(* Visualisation visuTimetable
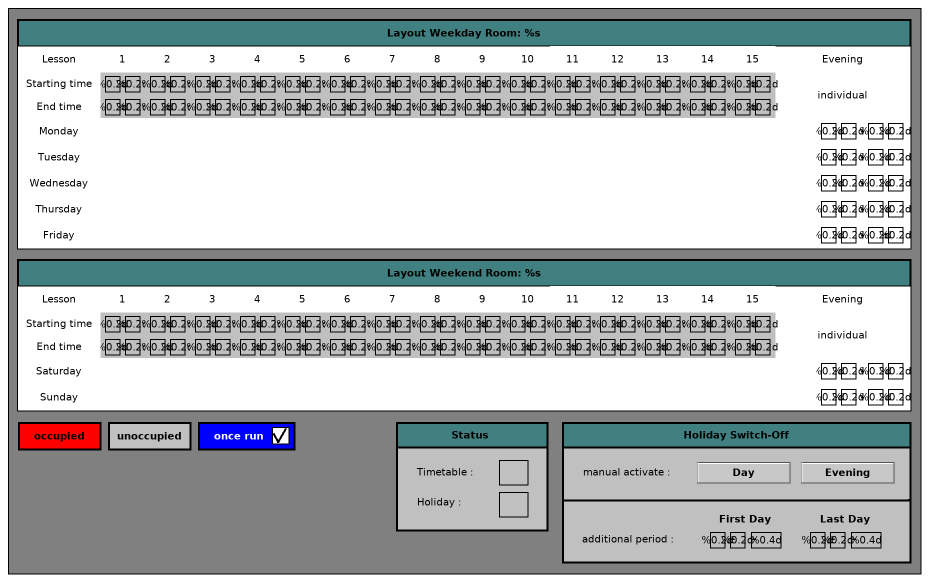
rectangle at (700,518)-(780,543): text "-     -"; tooltip First day Input format: DD-HH-YYYY
rectangle at (92,162)-(137,188): alarm colour if $typTimetable$.wDayLesson[3].1; toggles $typTimetable$.wDayLesson[3].1
rectangle at (137,162)-(182,188): alarm colour if $typTimetable$.wDayLesson[3].2; toggles $typTimetable$.wDayLesson[3].2
rectangle at (182,162)-(227,188): alarm colour if $typTimetable$.wDayLesson[3].3; toggles $typTimetable$.wDayLesson[3].3
rectangle at (227,162)-(272,188): alarm colour if $typTimetable$.wDayLesson[3].4; toggles $typTimetable$.wDayLesson[3].4
rectangle at (272,162)-(317,188): alarm colour if $typTimetable$.wDayLesson[3].5; toggles $typTimetable$.wDayLesson[3].5
rectangle at (317,162)-(362,188): alarm colour if $typTimetable$.wDayLesson[3].6; toggles $typTimetable$.wDayLesson[3].6
rectangle at (362,162)-(407,188): alarm colour if $typTimetable$.wDayLesson[3].7; toggles $typTimetable$.wDayLesson[3].7
rectangle at (407,162)-(452,188): alarm colour if $typTimetable$.wDayLesson[3].8; toggles $typTimetable$.wDayLesson[3].8
rectangle at (452,162)-(497,188): alarm colour if $typTimetable$.wDayLesson[3].9; toggles $typTimetable$.wDayLesson[3].9
rectangle at (497,162)-(542,188): alarm colour if $typTimetable$.wDayLesson[3].10; toggles $typTimetable$.wDayLesson[3].10
rectangle at (808,110)-(853,136): text ":"; tooltip Switch ON time of the scheduler single weekly
rectangle at (855,110)-(900,136): text ":"; tooltip Switch ON time of the scheduler single weekly
rectangle at (808,136)-(853,162): text ":"; tooltip Switch ON time of the scheduler single weekly
rectangle at (855,136)-(900,162): text ":"; tooltip Switch ON time of the scheduler single weekly
rectangle at (808,162)-(853,188): text ":"; tooltip Switch ON time of the scheduler single weekly
rectangle at (855,162)-(900,188): text ":"; tooltip Switch ON time of the scheduler single weekly
rectangle at (808,188)-(853,214): text ":"; tooltip Switch ON time of the scheduler single weekly
rectangle at (855,188)-(900,214): text ":"; tooltip Switch ON time of the scheduler single weekly
rectangle at (808,214)-(853,240): text ":"; tooltip Switch ON time of the scheduler single weekly
rectangle at (808,350)-(853,376): text ":"; tooltip Switch ON time of the scheduler single weekly
rectangle at (855,350)-(900,376): text ":"; tooltip Switch ON time of the scheduler single weekly
rectangle at (808,376)-(853,402): text ":"; tooltip Switch ON time of the scheduler single weekly
rectangle at (855,376)-(900,402): text ":"; tooltip Switch ON time of the scheduler single weekly
rectangle at (92,64)-(137,87): text ":"; tooltip Switch ON time
rectangle at (97,68)-(112,84): text "%0.2d"; shows $typLesson$.wWeekdayOn_hour[1]
rectangle at (117,68)-(132,84): text "%0.2d"; shows $typLesson$.wWeekdayOn_Minute[1]
rectangle at (137,64)-(182,87): text ":"; tooltip Switch ON time
rectangle at (142,68)-(157,84): text "%0.2d"; shows $typLesson$.wWeekdayOn_hour[2]
rectangle at (162,68)-(177,84): text "%0.2d"; shows $typLesson$.wWeekdayOn_Minute[2]
rectangle at (182,64)-(227,87): text ":"; tooltip Switch ON time
rectangle at (187,68)-(202,84): text "%0.2d"; shows $typLesson$.wWeekdayOn_hour[3]
rectangle at (207,68)-(222,84): text "%0.2d"; shows $typLesson$.wWeekdayOn_Minute[3]
rectangle at (227,64)-(272,87): text ":"; tooltip Switch ON time
rectangle at (232,68)-(247,84): text "%0.2d"; shows $typLesson$.wWeekdayOn_hour[4]
rectangle at (252,68)-(267,84): text "%0.2d"; shows $typLesson$.wWeekdayOn_Minute[4]
rectangle at (272,64)-(317,87): text ":"; tooltip Switch ON time
rectangle at (277,68)-(292,84): text "%0.2d"; shows $typLesson$.wWeekdayOn_hour[5]
rectangle at (297,68)-(312,84): text "%0.2d"; shows $typLesson$.wWeekdayOn_Minute[5]
rectangle at (317,64)-(362,87): text ":"; tooltip Switch ON time
rectangle at (322,68)-(337,84): text "%0.2d"; shows $typLesson$.wWeekdayOn_hour[6]
rectangle at (342,68)-(357,84): text "%0.2d"; shows $typLesson$.wWeekdayOn_Minute[6]
rectangle at (362,64)-(407,87): text ":"; tooltip Switch ON time
rectangle at (367,68)-(382,84): text "%0.2d"; shows $typLesson$.wWeekdayOn_hour[7]
rectangle at (387,68)-(402,84): text "%0.2d"; shows $typLesson$.wWeekdayOn_Minute[7]
rectangle at (407,64)-(452,87): text ":"; tooltip Switch ON time
rectangle at (412,68)-(427,84): text "%0.2d"; shows $typLesson$.wWeekdayOn_hour[8]
rectangle at (432,68)-(447,84): text "%0.2d"; shows $typLesson$.wWeekdayOn_Minute[8]
rectangle at (452,64)-(497,87): text ":"; tooltip Switch ON time
rectangle at (457,68)-(472,84): text "%0.2d"; shows $typLesson$.wWeekdayOn_hour[9]
rectangle at (477,68)-(492,84): text "%0.2d"; shows $typLesson$.wWeekdayOn_Minute[9]
rectangle at (497,64)-(542,87): text ":"; tooltip Switch ON time
rectangle at (502,68)-(517,84): text "%0.2d"; shows $typLesson$.wWeekdayOn_hour[10]
rectangle at (522,68)-(537,84): text "%0.2d"; shows $typLesson$.wWeekdayOn_Minute[10]
rectangle at (92,188)-(137,214): alarm colour if $typTimetable$.wDayLesson[4].1; toggles $typTimetable$.wDayLesson[4].1
rectangle at (137,188)-(182,214): alarm colour if $typTimetable$.wDayLesson[4].2; toggles $typTimetable$.wDayLesson[4].2
rectangle at (182,188)-(227,214): alarm colour if $typTimetable$.wDayLesson[4].3; toggles $typTimetable$.wDayLesson[4].3
rectangle at (227,188)-(272,214): alarm colour if $typTimetable$.wDayLesson[4].4; toggles $typTimetable$.wDayLesson[4].4
rectangle at (272,188)-(317,214): alarm colour if $typTimetable$.wDayLesson[4].5; toggles $typTimetable$.wDayLesson[4].5
rectangle at (317,188)-(362,214): alarm colour if $typTimetable$.wDayLesson[4].6; toggles $typTimetable$.wDayLesson[4].6
rectangle at (362,188)-(407,214): alarm colour if $typTimetable$.wDayLesson[4].7; toggles $typTimetable$.wDayLesson[4].7
rectangle at (407,188)-(452,214): alarm colour if $typTimetable$.wDayLesson[4].8; toggles $typTimetable$.wDayLesson[4].8
rectangle at (452,188)-(497,214): alarm colour if $typTimetable$.wDayLesson[4].9; toggles $typTimetable$.wDayLesson[4].9
rectangle at (497,188)-(542,214): alarm colour if $typTimetable$.wDayLesson[4].10; toggles $typTimetable$.wDayLesson[4].10
rectangle at (807,188)-(902,214): text "-"
rectangle at (807,214)-(902,240): text "-"
rectangle at (807,162)-(902,188): text "-"
rectangle at (807,136)-(902,162): text "-"
rectangle at (807,110)-(902,136): text "-"
rectangle at (813,115)-(828,131): text "%0.2d"; shows $typTimetable$.wEveningOn_hour[1]; editable 0..23
rectangle at (833,115)-(848,131): text "%0.2d"; shows $typTimetable$.wEveningOn_minute[1]; editable 0..59
rectangle at (860,115)-(875,131): text "%0.2d"; shows $typTimetable$.wEveningOff_hour[1]; editable 0..23
rectangle at (880,115)-(895,131): text "%0.2d"; shows $typTimetable$.wEveningOff_minute[1]; editable 0..59
rectangle at (813,141)-(828,157): text "%0.2d"; shows $typTimetable$.wEveningOn_hour[2]; editable 0..23
rectangle at (833,141)-(848,157): text "%0.2d"; shows $typTimetable$.wEveningOn_minute[2]; editable 0..59
rectangle at (860,141)-(875,157): text "%0.2d"; shows $typTimetable$.wEveningOff_hour[2]; editable 0..23
rectangle at (880,141)-(895,157): text "%0.2d"; shows $typTimetable$.wEveningOff_minute[2]; editable 0..59
rectangle at (813,193)-(828,209): text "%0.2d"; shows $typTimetable$.wEveningOn_hour[4]; editable 0..23
rectangle at (833,193)-(848,209): text "%0.2d"; shows $typTimetable$.wEveningOn_minute[4]; editable 0..59
rectangle at (860,193)-(875,209): text "%0.2d"; shows $typTimetable$.wEveningOff_hour[4]; editable 0..23
rectangle at (880,193)-(895,209): text "%0.2d"; shows $typTimetable$.wEveningOff_minute[4]; editable 0..59
rectangle at (813,219)-(828,235): text "%0.2d"; shows $typTimetable$.wEveningOn_hour[5]; editable 0..23
rectangle at (833,219)-(848,235): text "%0.2d"; shows $typTimetable$.wEveningOn_minute[5]; editable 0..59
rectangle at (813,167)-(828,183): text "%0.2d"; shows $typTimetable$.wEveningOn_hour[3]; editable 0..23
rectangle at (833,167)-(848,183): text "%0.2d"; shows $typTimetable$.wEveningOn_minute[3]; editable 0..59
rectangle at (860,167)-(875,183): text "%0.2d"; shows $typTimetable$.wEveningOff_hour[3]; editable 0..23
rectangle at (880,167)-(895,183): text "%0.2d"; shows $typTimetable$.wEveningOff_minute[3]; editable 0..59
rectangle at (807,350)-(902,376): text "-"
rectangle at (807,376)-(902,402): text "-"
rectangle at (813,355)-(828,371): text "%0.2d"; shows $typTimetable$.wEveningOn_hour[6]; editable 0..23
rectangle at (833,355)-(848,371): text "%0.2d"; shows $typTimetable$.wEveningOn_minute[6]; editable 0..59
rectangle at (860,355)-(875,371): text "%0.2d"; shows $typTimetable$.wEveningOff_hour[6]; editable 0..23
rectangle at (880,355)-(895,371): text "%0.2d"; shows $typTimetable$.wEveningOff_minute[6]; editable 0..59
rectangle at (813,381)-(828,397): text "%0.2d"; shows $typTimetable$.wEveningOn_hour[7]; editable 0..23
rectangle at (833,381)-(848,397): text "%0.2d"; shows $typTimetable$.wEveningOn_minute[7]; editable 0..59
rectangle at (860,381)-(875,397): text "%0.2d"; shows $typTimetable$.wEveningOff_hour[7]; editable 0..23
rectangle at (880,381)-(895,397): text "%0.2d"; shows $typTimetable$.wEveningOff_minute[7]; editable 0..59
rectangle at (92,110)-(137,136): alarm colour if $typTimetable$.wDayLesson[1].1; toggles $typTimetable$.wDayLesson[1].1
rectangle at (137,110)-(182,136): alarm colour if $typTimetable$.wDayLesson[1].2; toggles $typTimetable$.wDayLesson[1].2
rectangle at (182,110)-(227,136): alarm colour if $typTimetable$.wDayLesson[1].3; toggles $typTimetable$.wDayLesson[1].3
rectangle at (227,110)-(272,136): alarm colour if $typTimetable$.wDayLesson[1].4; toggles $typTimetable$.wDayLesson[1].4
rectangle at (272,110)-(317,136): alarm colour if $typTimetable$.wDayLesson[1].5; toggles $typTimetable$.wDayLesson[1].5
rectangle at (317,110)-(362,136): alarm colour if $typTimetable$.wDayLesson[1].6; toggles $typTimetable$.wDayLesson[1].6
rectangle at (362,110)-(407,136): alarm colour if $typTimetable$.wDayLesson[1].7; toggles $typTimetable$.wDayLesson[1].7
rectangle at (407,110)-(452,136): alarm colour if $typTimetable$.wDayLesson[1].8; toggles $typTimetable$.wDayLesson[1].8
rectangle at (452,110)-(497,136): alarm colour if $typTimetable$.wDayLesson[1].9; toggles $typTimetable$.wDayLesson[1].9
rectangle at (497,110)-(542,136): alarm colour if $typTimetable$.wDayLesson[1].10; toggles $typTimetable$.wDayLesson[1].10
rectangle at (92,136)-(137,162): alarm colour if $typTimetable$.wDayLesson[2].1; toggles $typTimetable$.wDayLesson[2].1
rectangle at (137,136)-(182,162): alarm colour if $typTimetable$.wDayLesson[2].2; toggles $typTimetable$.wDayLesson[2].2
rectangle at (182,136)-(227,162): alarm colour if $typTimetable$.wDayLesson[2].3; toggles $typTimetable$.wDayLesson[2].3
rectangle at (227,136)-(272,162): alarm colour if $typTimetable$.wDayLesson[2].4; toggles $typTimetable$.wDayLesson[2].4
rectangle at (272,136)-(317,162): alarm colour if $typTimetable$.wDayLesson[2].5; toggles $typTimetable$.wDayLesson[2].5
rectangle at (317,136)-(362,162): alarm colour if $typTimetable$.wDayLesson[2].6; toggles $typTimetable$.wDayLesson[2].6
rectangle at (362,136)-(407,162): alarm colour if $typTimetable$.wDayLesson[2].7; toggles $typTimetable$.wDayLesson[2].7
rectangle at (407,136)-(452,162): alarm colour if $typTimetable$.wDayLesson[2].8; toggles $typTimetable$.wDayLesson[2].8
rectangle at (452,136)-(497,162): alarm colour if $typTimetable$.wDayLesson[2].9; toggles $typTimetable$.wDayLesson[2].9
rectangle at (497,136)-(542,162): alarm colour if $typTimetable$.wDayLesson[2].10; toggles $typTimetable$.wDayLesson[2].10
rectangle at (92,214)-(137,240): alarm colour if $typTimetable$.wDayLesson[5].1; toggles $typTimetable$.wDayLesson[5].1
rectangle at (137,214)-(182,240): alarm colour if $typTimetable$.wDayLesson[5].2; toggles $typTimetable$.wDayLesson[5].2
rectangle at (182,214)-(227,240): alarm colour if $typTimetable$.wDayLesson[5].3; toggles $typTimetable$.wDayLesson[5].3
rectangle at (227,214)-(272,240): alarm colour if $typTimetable$.wDayLesson[5].4; toggles $typTimetable$.wDayLesson[5].4
rectangle at (272,214)-(317,240): alarm colour if $typTimetable$.wDayLesson[5].5; toggles $typTimetable$.wDayLesson[5].5
rectangle at (317,214)-(362,240): alarm colour if $typTimetable$.wDayLesson[5].6; toggles $typTimetable$.wDayLesson[5].6
rectangle at (362,214)-(407,240): alarm colour if $typTimetable$.wDayLesson[5].7; toggles $typTimetable$.wDayLesson[5].7
rectangle at (407,214)-(452,240): alarm colour if $typTimetable$.wDayLesson[5].8; toggles $typTimetable$.wDayLesson[5].8
rectangle at (452,214)-(497,240): alarm colour if $typTimetable$.wDayLesson[5].9; toggles $typTimetable$.wDayLesson[5].9
rectangle at (497,214)-(542,240): alarm colour if $typTimetable$.wDayLesson[5].10; toggles $typTimetable$.wDayLesson[5].10
rectangle at (92,350)-(137,376): alarm colour if $typTimetable$.wDayLesson[6].1; toggles $typTimetable$.wDayLesson[6].1
rectangle at (137,350)-(182,376): alarm colour if $typTimetable$.wDayLesson[6].2; toggles $typTimetable$.wDayLesson[6].2
rectangle at (182,350)-(227,376): alarm colour if $typTimetable$.wDayLesson[6].3; toggles $typTimetable$.wDayLesson[6].3
rectangle at (227,350)-(272,376): alarm colour if $typTimetable$.wDayLesson[6].4; toggles $typTimetable$.wDayLesson[6].4
rectangle at (272,350)-(317,376): alarm colour if $typTimetable$.wDayLesson[6].5; toggles $typTimetable$.wDayLesson[6].5
rectangle at (317,350)-(362,376): alarm colour if $typTimetable$.wDayLesson[6].6; toggles $typTimetable$.wDayLesson[6].6
rectangle at (362,350)-(407,376): alarm colour if $typTimetable$.wDayLesson[6].7; toggles $typTimetable$.wDayLesson[6].7
rectangle at (407,350)-(452,376): alarm colour if $typTimetable$.wDayLesson[6].8; toggles $typTimetable$.wDayLesson[6].8
rectangle at (452,350)-(497,376): alarm colour if $typTimetable$.wDayLesson[6].9; toggles $typTimetable$.wDayLesson[6].9
rectangle at (497,350)-(542,376): alarm colour if $typTimetable$.wDayLesson[6].10; toggles $typTimetable$.wDayLesson[6].10
rectangle at (92,376)-(137,402): alarm colour if $typTimetable$.wDayLesson[7].1; toggles $typTimetable$.wDayLesson[7].1
rectangle at (137,376)-(182,402): alarm colour if $typTimetable$.wDayLesson[7].2; toggles $typTimetable$.wDayLesson[7].2
rectangle at (182,376)-(227,402): alarm colour if $typTimetable$.wDayLesson[7].3; toggles $typTimetable$.wDayLesson[7].3
rectangle at (227,376)-(272,402): alarm colour if $typTimetable$.wDayLesson[7].4; toggles $typTimetable$.wDayLesson[7].4
rectangle at (272,376)-(317,402): alarm colour if $typTimetable$.wDayLesson[7].5; toggles $typTimetable$.wDayLesson[7].5
rectangle at (317,376)-(362,402): alarm colour if $typTimetable$.wDayLesson[7].6; toggles $typTimetable$.wDayLesson[7].6
rectangle at (362,376)-(407,402): alarm colour if $typTimetable$.wDayLesson[7].7; toggles $typTimetable$.wDayLesson[7].7
rectangle at (407,376)-(452,402): alarm colour if $typTimetable$.wDayLesson[7].8; toggles $typTimetable$.wDayLesson[7].8
rectangle at (452,376)-(497,402): alarm colour if $typTimetable$.wDayLesson[7].9; toggles $typTimetable$.wDayLesson[7].9
rectangle at (497,376)-(542,402): alarm colour if $typTimetable$.wDayLesson[7].10; toggles $typTimetable$.wDayLesson[7].10
rectangle at (92,87)-(137,110): text ":"; tooltip Switch OFF time
rectangle at (97,91)-(112,107): text "%0.2d"; shows $typLesson$.wWeekdayOff_hour[1]
rectangle at (117,91)-(132,107): text "%0.2d"; shows $typLesson$.wWeekdayOff_Minute[1]
rectangle at (137,87)-(182,110): text ":"; tooltip Switch OFF time
rectangle at (142,91)-(157,107): text "%0.2d"; shows $typLesson$.wWeekdayOff_hour[2]
rectangle at (162,91)-(177,107): text "%0.2d"; shows $typLesson$.wWeekdayOff_Minute[2]
rectangle at (182,87)-(227,110): text ":"; tooltip Switch OFF time
rectangle at (187,91)-(202,107): text "%0.2d"; shows $typLesson$.wWeekdayOff_hour[3]
rectangle at (207,91)-(222,107): text "%0.2d"; shows $typLesson$.wWeekdayOff_Minute[3]
rectangle at (227,87)-(272,110): text ":"; tooltip Switch OFF time
rectangle at (232,91)-(247,107): text "%0.2d"; shows $typLesson$.wWeekdayOff_hour[4]
rectangle at (252,91)-(267,107): text "%0.2d"; shows $typLesson$.wWeekdayOff_Minute[4]
rectangle at (272,87)-(317,110): text ":"; tooltip Switch OFF time
rectangle at (277,91)-(292,107): text "%0.2d"; shows $typLesson$.wWeekdayOff_hour[5]
rectangle at (297,91)-(312,107): text "%0.2d"; shows $typLesson$.wWeekdayOff_Minute[5]
rectangle at (317,87)-(362,110): text ":"; tooltip Switch OFF time
rectangle at (322,91)-(337,107): text "%0.2d"; shows $typLesson$.wWeekdayOff_hour[6]
rectangle at (342,91)-(357,107): text "%0.2d"; shows $typLesson$.wWeekdayOff_Minute[6]
rectangle at (362,87)-(407,110): text ":"; tooltip Switch OFF time
rectangle at (367,91)-(382,107): text "%0.2d"; shows $typLesson$.wWeekdayOff_hour[7]
rectangle at (387,91)-(402,107): text "%0.2d"; shows $typLesson$.wWeekdayOff_Minute[7]
rectangle at (407,87)-(452,110): text ":"; tooltip Switch OFF time
rectangle at (412,91)-(427,107): text "%0.2d"; shows $typLesson$.wWeekdayOff_hour[8]
rectangle at (432,91)-(447,107): text "%0.2d"; shows $typLesson$.wWeekdayOff_Minute[8]
rectangle at (452,87)-(497,110): text ":"; tooltip Switch OFF time
rectangle at (457,91)-(472,107): text "%0.2d"; shows $typLesson$.wWeekdayOff_hour[9]
rectangle at (477,91)-(492,107): text "%0.2d"; shows $typLesson$.wWeekdayOff_Minute[9]
rectangle at (497,87)-(542,110): text ":"; tooltip Switch OFF time
rectangle at (502,91)-(517,107): text "%0.2d"; shows $typLesson$.wWeekdayOff_hour[10]
rectangle at (522,91)-(537,107): text "%0.2d"; shows $typLesson$.wWeekdayOff_Minute[10]
rectangle at (767,64)-(902,110): text "individual"
rectangle at (92,38)-(137,64): text "1"
rectangle at (137,38)-(182,64): text "2"
rectangle at (182,38)-(227,64): text "3"
rectangle at (227,38)-(272,64): text "4"
rectangle at (272,38)-(317,64): text "5"
rectangle at (317,38)-(362,64): text "6"
rectangle at (362,38)-(407,64): text "7"
rectangle at (407,38)-(452,64): text "8"
rectangle at (452,38)-(497,64): text "9"
rectangle at (497,38)-(542,64): text "10"
rectangle at (767,38)-(902,64): text "Evening"
rectangle at (10,38)-(92,64): text "Lesson"
rectangle at (10,64)-(92,87): text "Starting time"
rectangle at (10,87)-(92,110): text "End time"
rectangle at (10,110)-(92,136): text "Monday"
rectangle at (10,136)-(92,162): text "Tuesday"
rectangle at (10,162)-(92,188): text "Wednesday"
rectangle at (10,188)-(92,214): text "Thursday"
rectangle at (10,214)-(92,240): text "Friday"
rectangle at (10,350)-(92,376): text "Saturday"
rectangle at (10,376)-(92,402): text "Sunday"
rectangle at (92,304)-(137,327): text ":"; tooltip Switch ON time
rectangle at (97,308)-(112,324): text "%0.2d"; shows $typLesson$.wWeekendOn_hour[1]
rectangle at (117,308)-(132,324): text "%0.2d"; shows $typLesson$.wWeekendOn_Minute[1]
rectangle at (137,304)-(182,327): text ":"; tooltip Switch ON time
rectangle at (142,308)-(157,324): text "%0.2d"; shows $typLesson$.wWeekendOn_hour[2]
rectangle at (162,308)-(177,324): text "%0.2d"; shows $typLesson$.wWeekendOn_Minute[2]
rectangle at (182,304)-(227,327): text ":"; tooltip Switch ON time
rectangle at (187,308)-(202,324): text "%0.2d"; shows $typLesson$.wWeekendOn_hour[3]
rectangle at (207,308)-(222,324): text "%0.2d"; shows $typLesson$.wWeekendOn_Minute[3]
rectangle at (227,304)-(272,327): text ":"; tooltip Switch ON time
rectangle at (232,308)-(247,324): text "%0.2d"; shows $typLesson$.wWeekendOn_hour[4]
rectangle at (252,308)-(267,324): text "%0.2d"; shows $typLesson$.wWeekendOn_Minute[4]
rectangle at (272,304)-(317,327): text ":"; tooltip Switch ON time
rectangle at (277,308)-(292,324): text "%0.2d"; shows $typLesson$.wWeekendOn_hour[5]
rectangle at (297,308)-(312,324): text "%0.2d"; shows $typLesson$.wWeekendOn_Minute[5]
rectangle at (317,304)-(362,327): text ":"; tooltip Switch ON time
rectangle at (322,308)-(337,324): text "%0.2d"; shows $typLesson$.wWeekendOn_hour[6]
rectangle at (342,308)-(357,324): text "%0.2d"; shows $typLesson$.wWeekendOn_Minute[6]
rectangle at (362,304)-(407,327): text ":"; tooltip Switch ON time
rectangle at (367,308)-(382,324): text "%0.2d"; shows $typLesson$.wWeekendOn_hour[7]
rectangle at (387,308)-(402,324): text "%0.2d"; shows $typLesson$.wWeekendOn_Minute[7]
rectangle at (407,304)-(452,327): text ":"; tooltip Switch ON time
rectangle at (412,308)-(427,324): text "%0.2d"; shows $typLesson$.wWeekendOn_hour[8]
rectangle at (432,308)-(447,324): text "%0.2d"; shows $typLesson$.wWeekendOn_Minute[8]
rectangle at (452,304)-(497,327): text ":"; tooltip Switch ON time
rectangle at (457,308)-(472,324): text "%0.2d"; shows $typLesson$.wWeekendOn_hour[9]
rectangle at (477,308)-(492,324): text "%0.2d"; shows $typLesson$.wWeekendOn_Minute[9]
rectangle at (497,304)-(542,327): text ":"; tooltip Switch ON time
rectangle at (502,308)-(517,324): text "%0.2d"; shows $typLesson$.wWeekendOn_hour[10]
rectangle at (522,308)-(537,324): text "%0.2d"; shows $typLesson$.wWeekendOn_Minute[10]
rectangle at (92,327)-(137,350): text ":"; tooltip Switch OFF time
rectangle at (97,331)-(112,347): text "%0.2d"; shows $typLesson$.wWeekendOff_hour[1]
rectangle at (117,331)-(132,347): text "%0.2d"; shows $typLesson$.wWeekendOff_Minute[1]
rectangle at (137,327)-(182,350): text ":"; tooltip Switch OFF time
rectangle at (142,331)-(157,347): text "%0.2d"; shows $typLesson$.wWeekendOff_hour[2]
rectangle at (162,331)-(177,347): text "%0.2d"; shows $typLesson$.wWeekendOff_Minute[2]
rectangle at (182,327)-(227,350): text ":"; tooltip Switch OFF time
rectangle at (187,331)-(202,347): text "%0.2d"; shows $typLesson$.wWeekendOff_hour[3]
rectangle at (207,331)-(222,347): text "%0.2d"; shows $typLesson$.wWeekendOff_Minute[3]
rectangle at (227,327)-(272,350): text ":"; tooltip Switch OFF time
rectangle at (232,331)-(247,347): text "%0.2d"; shows $typLesson$.wWeekendOff_hour[4]
rectangle at (252,331)-(267,347): text "%0.2d"; shows $typLesson$.wWeekendOff_Minute[4]
rectangle at (272,327)-(317,350): text ":"; tooltip Switch OFF time
rectangle at (277,331)-(292,347): text "%0.2d"; shows $typLesson$.wWeekendOff_hour[5]
rectangle at (297,331)-(312,347): text "%0.2d"; shows $typLesson$.wWeekendOff_Minute[5]
rectangle at (317,327)-(362,350): text ":"; tooltip Switch OFF time
rectangle at (322,331)-(337,347): text "%0.2d"; shows $typLesson$.wWeekendOff_hour[6]
rectangle at (342,331)-(357,347): text "%0.2d"; shows $typLesson$.wWeekendOff_Minute[6]
rectangle at (362,327)-(407,350): text ":"; tooltip Switch OFF time
rectangle at (367,331)-(382,347): text "%0.2d"; shows $typLesson$.wWeekendOff_hour[7]
rectangle at (387,331)-(402,347): text "%0.2d"; shows $typLesson$.wWeekendOff_Minute[7]
rectangle at (407,327)-(452,350): text ":"; tooltip Switch OFF time
rectangle at (412,331)-(427,347): text "%0.2d"; shows $typLesson$.wWeekendOff_hour[8]
rectangle at (432,331)-(447,347): text "%0.2d"; shows $typLesson$.wWeekendOff_Minute[8]
rectangle at (452,327)-(497,350): text ":"; tooltip Switch OFF time
rectangle at (457,331)-(472,347): text "%0.2d"; shows $typLesson$.wWeekendOff_hour[9]
rectangle at (477,331)-(492,347): text "%0.2d"; shows $typLesson$.wWeekendOff_Minute[9]
rectangle at (497,327)-(542,350): text ":"; tooltip Switch OFF time
rectangle at (502,331)-(517,347): text "%0.2d"; shows $typLesson$.wWeekendOff_hour[10]
rectangle at (522,331)-(537,347): text "%0.2d"; shows $typLesson$.wWeekendOff_Minute[10]
rectangle at (767,304)-(902,350): text "individual"
rectangle at (92,278)-(137,304): text "1"
rectangle at (137,278)-(182,304): text "2"
rectangle at (182,278)-(227,304): text "3"
rectangle at (227,278)-(272,304): text "4"
rectangle at (272,278)-(317,304): text "5"
rectangle at (317,278)-(362,304): text "6"
rectangle at (362,278)-(407,304): text "7"
rectangle at (407,278)-(452,304): text "8"
rectangle at (452,278)-(497,304): text "9"
rectangle at (497,278)-(542,304): text "10"
rectangle at (767,278)-(902,304): text "Evening"
rectangle at (10,278)-(92,304): text "Lesson"
rectangle at (10,304)-(92,327): text "Starting time"
rectangle at (10,327)-(92,350): text "End time"
rectangle at (10,252)-(902,278): text "Layout Weekend Room: %s"; shows $typTimetable$.stRoomNr; editable
rectangle at (10,12)-(902,38): text "Layout Weekday Room: %s"; shows $typTimetable$.stRoomNr; editable
button at (689,454)-(782,475): text "Day"; toggles $typTimetable$.bConfig.0
button at (793,454)-(886,475): text "Evening"; toggles $typTimetable$.bConfig.1
rectangle at (554,414)-(903,440): text "Holiday Switch-Off"
rectangle at (10,414)-(93,442): text "occupied"
rectangle at (100,414)-(183,442): text "unoccupied"
rectangle at (542,162)-(587,188): alarm colour if $typTimetable$.wDayLesson[3].11; toggles $typTimetable$.wDayLesson[3].11
rectangle at (542,64)-(587,87): text ":"; tooltip Switch ON time
rectangle at (547,68)-(562,84): text "%0.2d"; shows $typLesson$.wWeekdayOn_hour[11]
rectangle at (567,68)-(582,84): text "%0.2d"; shows $typLesson$.wWeekdayOn_Minute[11]
rectangle at (542,188)-(587,214): alarm colour if $typTimetable$.wDayLesson[4].11; toggles $typTimetable$.wDayLesson[4].11
rectangle at (542,110)-(587,136): alarm colour if $typTimetable$.wDayLesson[1].11; toggles $typTimetable$.wDayLesson[1].11
rectangle at (542,136)-(587,162): alarm colour if $typTimetable$.wDayLesson[2].11; toggles $typTimetable$.wDayLesson[2].11
rectangle at (542,214)-(587,240): alarm colour if $typTimetable$.wDayLesson[5].11; toggles $typTimetable$.wDayLesson[5].11
rectangle at (542,87)-(587,110): text ":"; tooltip Switch OFF time
rectangle at (547,91)-(562,107): text "%0.2d"; shows $typLesson$.wWeekdayOff_hour[11]
rectangle at (567,91)-(582,107): text "%0.2d"; shows $typLesson$.wWeekdayOff_Minute[11]
rectangle at (542,38)-(587,64): text "11"
rectangle at (587,162)-(632,188): alarm colour if $typTimetable$.wDayLesson[3].12; toggles $typTimetable$.wDayLesson[3].12
rectangle at (587,64)-(632,87): text ":"; tooltip Switch ON time
rectangle at (592,68)-(607,84): text "%0.2d"; shows $typLesson$.wWeekdayOn_hour[12]
rectangle at (612,68)-(627,84): text "%0.2d"; shows $typLesson$.wWeekdayOn_Minute[12]
rectangle at (587,188)-(632,214): alarm colour if $typTimetable$.wDayLesson[4].12; toggles $typTimetable$.wDayLesson[4].12
rectangle at (587,110)-(632,136): alarm colour if $typTimetable$.wDayLesson[1].12; toggles $typTimetable$.wDayLesson[1].12
rectangle at (587,136)-(632,162): alarm colour if $typTimetable$.wDayLesson[2].12; toggles $typTimetable$.wDayLesson[2].12
rectangle at (587,214)-(632,240): alarm colour if $typTimetable$.wDayLesson[5].12; toggles $typTimetable$.wDayLesson[5].12
rectangle at (587,87)-(632,110): text ":"; tooltip Switch OFF time
rectangle at (592,91)-(607,107): text "%0.2d"; shows $typLesson$.wWeekdayOff_hour[12]
rectangle at (612,91)-(627,107): text "%0.2d"; shows $typLesson$.wWeekdayOff_Minute[12]
rectangle at (587,38)-(632,64): text "12"
rectangle at (632,162)-(677,188): alarm colour if $typTimetable$.wDayLesson[3].13; toggles $typTimetable$.wDayLesson[3].13
rectangle at (632,64)-(677,87): text ":"; tooltip Switch ON time
rectangle at (637,68)-(652,84): text "%0.2d"; shows $typLesson$.wWeekdayOn_hour[13]
rectangle at (657,68)-(672,84): text "%0.2d"; shows $typLesson$.wWeekdayOn_Minute[13]
rectangle at (632,188)-(677,214): alarm colour if $typTimetable$.wDayLesson[4].13; toggles $typTimetable$.wDayLesson[4].13
rectangle at (632,110)-(677,136): alarm colour if $typTimetable$.wDayLesson[1].13; toggles $typTimetable$.wDayLesson[1].13
rectangle at (632,136)-(677,162): alarm colour if $typTimetable$.wDayLesson[2].13; toggles $typTimetable$.wDayLesson[2].13
rectangle at (632,214)-(677,240): alarm colour if $typTimetable$.wDayLesson[5].13; toggles $typTimetable$.wDayLesson[5].13
rectangle at (632,87)-(677,110): text ":"; tooltip Switch OFF time
rectangle at (637,91)-(652,107): text "%0.2d"; shows $typLesson$.wWeekdayOff_hour[13]
rectangle at (657,91)-(672,107): text "%0.2d"; shows $typLesson$.wWeekdayOff_Minute[13]
rectangle at (632,38)-(677,64): text "13"
rectangle at (677,162)-(722,188): alarm colour if $typTimetable$.wDayLesson[3].14; toggles $typTimetable$.wDayLesson[3].14
rectangle at (677,64)-(722,87): text ":"; tooltip Switch ON time
rectangle at (682,68)-(697,84): text "%0.2d"; shows $typLesson$.wWeekdayOn_hour[14]
rectangle at (702,68)-(717,84): text "%0.2d"; shows $typLesson$.wWeekdayOn_Minute[14]
rectangle at (677,188)-(722,214): alarm colour if $typTimetable$.wDayLesson[4].14; toggles $typTimetable$.wDayLesson[4].14
rectangle at (677,110)-(722,136): alarm colour if $typTimetable$.wDayLesson[1].14; toggles $typTimetable$.wDayLesson[1].14
rectangle at (677,136)-(722,162): alarm colour if $typTimetable$.wDayLesson[2].14; toggles $typTimetable$.wDayLesson[2].14
rectangle at (677,214)-(722,240): alarm colour if $typTimetable$.wDayLesson[5].14; toggles $typTimetable$.wDayLesson[5].14
rectangle at (677,87)-(722,110): text ":"; tooltip Switch OFF time
rectangle at (682,91)-(697,107): text "%0.2d"; shows $typLesson$.wWeekdayOff_hour[14]
rectangle at (702,91)-(717,107): text "%0.2d"; shows $typLesson$.wWeekdayOff_Minute[14]
rectangle at (677,38)-(722,64): text "14"
rectangle at (722,162)-(767,188): alarm colour if $typTimetable$.wDayLesson[3].15; toggles $typTimetable$.wDayLesson[3].15
rectangle at (722,64)-(767,87): text ":"; tooltip Switch ON time
rectangle at (727,68)-(742,84): text "%0.2d"; shows $typLesson$.wWeekdayOn_hour[15]
rectangle at (747,68)-(762,84): text "%0.2d"; shows $typLesson$.wWeekdayOn_Minute[15]
rectangle at (722,188)-(767,214): alarm colour if $typTimetable$.wDayLesson[4].15; toggles $typTimetable$.wDayLesson[4].15
rectangle at (722,110)-(767,136): alarm colour if $typTimetable$.wDayLesson[1].15; toggles $typTimetable$.wDayLesson[1].15
rectangle at (722,136)-(767,162): alarm colour if $typTimetable$.wDayLesson[2].15; toggles $typTimetable$.wDayLesson[2].15
rectangle at (722,214)-(767,240): alarm colour if $typTimetable$.wDayLesson[5].15; toggles $typTimetable$.wDayLesson[5].15
rectangle at (722,87)-(767,110): text ":"; tooltip Switch OFF time
rectangle at (727,91)-(742,107): text "%0.2d"; shows $typLesson$.wWeekdayOff_hour[15]
rectangle at (747,91)-(762,107): text "%0.2d"; shows $typLesson$.wWeekdayOff_Minute[15]
rectangle at (722,38)-(767,64): text "15"
rectangle at (542,350)-(587,376): alarm colour if $typTimetable$.wDayLesson[6].11; toggles $typTimetable$.wDayLesson[6].11
rectangle at (542,376)-(587,402): alarm colour if $typTimetable$.wDayLesson[7].11; toggles $typTimetable$.wDayLesson[7].11
rectangle at (542,304)-(587,327): text ":"; tooltip Switch ON time
rectangle at (547,308)-(562,324): text "%0.2d"; shows $typLesson$.wWeekendOn_hour[11]
rectangle at (567,308)-(582,324): text "%0.2d"; shows $typLesson$.wWeekendOn_Minute[11]
rectangle at (542,327)-(587,350): text ":"; tooltip Switch OFF time
rectangle at (547,331)-(562,347): text "%0.2d"; shows $typLesson$.wWeekendOff_hour[11]
rectangle at (567,331)-(582,347): text "%0.2d"; shows $typLesson$.wWeekendOff_Minute[11]
rectangle at (542,278)-(587,304): text "11"
rectangle at (587,350)-(632,376): alarm colour if $typTimetable$.wDayLesson[6].12; toggles $typTimetable$.wDayLesson[6].12
rectangle at (587,376)-(632,402): alarm colour if $typTimetable$.wDayLesson[7].12; toggles $typTimetable$.wDayLesson[7].12
rectangle at (587,304)-(632,327): text ":"; tooltip Switch ON time
rectangle at (592,308)-(607,324): text "%0.2d"; shows $typLesson$.wWeekendOn_hour[12]
rectangle at (612,308)-(627,324): text "%0.2d"; shows $typLesson$.wWeekendOn_Minute[12]
rectangle at (587,327)-(632,350): text ":"; tooltip Switch OFF time
rectangle at (592,331)-(607,347): text "%0.2d"; shows $typLesson$.wWeekendOff_hour[12]
rectangle at (612,331)-(627,347): text "%0.2d"; shows $typLesson$.wWeekendOff_Minute[12]
rectangle at (587,278)-(632,304): text "12"
rectangle at (632,350)-(677,376): alarm colour if $typTimetable$.wDayLesson[6].13; toggles $typTimetable$.wDayLesson[6].13
rectangle at (632,376)-(677,402): alarm colour if $typTimetable$.wDayLesson[7].13; toggles $typTimetable$.wDayLesson[7].13
rectangle at (632,304)-(677,327): text ":"; tooltip Switch ON time
rectangle at (637,308)-(652,324): text "%0.2d"; shows $typLesson$.wWeekendOn_hour[13]
rectangle at (657,308)-(672,324): text "%0.2d"; shows $typLesson$.wWeekendOn_Minute[13]
rectangle at (632,327)-(677,350): text ":"; tooltip Switch OFF time
rectangle at (637,331)-(652,347): text "%0.2d"; shows $typLesson$.wWeekendOff_hour[13]
rectangle at (657,331)-(672,347): text "%0.2d"; shows $typLesson$.wWeekendOff_Minute[13]
rectangle at (632,278)-(677,304): text "13"
rectangle at (677,350)-(722,376): alarm colour if $typTimetable$.wDayLesson[6].14; toggles $typTimetable$.wDayLesson[6].14
rectangle at (677,376)-(722,402): alarm colour if $typTimetable$.wDayLesson[7].14; toggles $typTimetable$.wDayLesson[7].14
rectangle at (677,304)-(722,327): text ":"; tooltip Switch ON time
rectangle at (682,308)-(697,324): text "%0.2d"; shows $typLesson$.wWeekendOn_hour[14]
rectangle at (702,308)-(717,324): text "%0.2d"; shows $typLesson$.wWeekendOn_Minute[14]
rectangle at (677,327)-(722,350): text ":"; tooltip Switch OFF time
rectangle at (682,331)-(697,347): text "%0.2d"; shows $typLesson$.wWeekendOff_hour[14]
rectangle at (702,331)-(717,347): text "%0.2d"; shows $typLesson$.wWeekendOff_Minute[14]
rectangle at (677,278)-(722,304): text "14"
rectangle at (722,350)-(767,376): alarm colour if $typTimetable$.wDayLesson[6].15; toggles $typTimetable$.wDayLesson[6].15
rectangle at (722,376)-(767,402): alarm colour if $typTimetable$.wDayLesson[7].15; toggles $typTimetable$.wDayLesson[7].15
rectangle at (722,304)-(767,327): text ":"; tooltip Switch ON time
rectangle at (727,308)-(742,324): text "%0.2d"; shows $typLesson$.wWeekendOn_hour[15]
rectangle at (747,308)-(762,324): text "%0.2d"; shows $typLesson$.wWeekendOn_Minute[15]
rectangle at (722,327)-(767,350): text ":"; tooltip Switch OFF time
rectangle at (727,331)-(742,347): text "%0.2d"; shows $typLesson$.wWeekendOff_hour[15]
rectangle at (747,331)-(762,347): text "%0.2d"; shows $typLesson$.wWeekendOff_Minute[15]
rectangle at (722,278)-(767,304): text "15"
rectangle at (767,110)-(807,136): alarm colour if $typTimetable$.wDayLesson[1].0; toggles $typTimetable$.wDayLesson[1].0
rectangle at (767,136)-(807,162): alarm colour if $typTimetable$.wDayLesson[2].0; toggles $typTimetable$.wDayLesson[2].0
rectangle at (767,162)-(807,188): alarm colour if $typTimetable$.wDayLesson[3].0; toggles $typTimetable$.wDayLesson[3].0
rectangle at (767,188)-(807,214): alarm colour if $typTimetable$.wDayLesson[4].0; toggles $typTimetable$.wDayLesson[4].0
rectangle at (767,214)-(807,240): alarm colour if $typTimetable$.wDayLesson[5].0; toggles $typTimetable$.wDayLesson[5].0
rectangle at (767,350)-(807,376): alarm colour if $typTimetable$.wDayLesson[6].0; toggles $typTimetable$.wDayLesson[6].0
rectangle at (767,376)-(807,402): alarm colour if $typTimetable$.wDayLesson[7].0; toggles $typTimetable$.wDayLesson[7].0
rectangle at (800,518)-(880,543): text "-     -"; tooltip Last day Input format: DD-HH-YYYY
rectangle at (802,524)-(817,540): text "%0.2d"; shows $typTimetable$.wSpecialLastDay[1]; editable 0..31
rectangle at (822,524)-(837,540): text "%0.2d"; shows $typTimetable$.wSpecialLastDay[2]; editable 0..12
rectangle at (843,524)-(873,540): text "%0.4d"; shows $typTimetable$.wSpecialLastDay[3]; editable 0..2099
rectangle at (702,524)-(717,540): text "%0.2d"; shows $typTimetable$.wSpecialFirstDay[1]; editable 0..31
rectangle at (722,524)-(737,540): text "%0.2d"; shows $typTimetable$.wSpecialFirstDay[2]; editable 0..12
rectangle at (743,524)-(773,540): text "%0.4d"; shows $typTimetable$.wSpecialFirstDay[3]; editable 0..2099
rectangle at (388,414)-(540,440): text "Status"
rectangle at (395,451)-(480,477): text "Timetable :"
rectangle at (395,481)-(473,507): text "Holiday :"
rectangle at (561,451)-(689,477): text "manual activate :"
rectangle at (560,518)-(688,544): text "additional period :"
rectangle at (697,499)-(777,523): text "First Day"
rectangle at (797,499)-(877,523): text "Last Day"
rectangle at (491,452)-(520,477): alarm colour if $typTimetable$.bStatus.1
rectangle at (491,484)-(520,509): alarm colour if $typTimetable$.bStatus.2
rectangle at (92,110)-(137,136): invisible if NOT $typTimetable$.bConfig.2 AND NOT ($typTimetable$.wDayLessonOnce[1].1 AND NOT $typTimetable$.bConfig.2); alarm colour if $typTimetable$.wDayLessonOnce[1].1; toggles $typTimetable$.wDayLessonOnce[1].1
rectangle at (137,110)-(182,136): invisible if NOT $typTimetable$.bConfig.2 AND NOT ($typTimetable$.wDayLessonOnce[1].2 AND NOT $typTimetable$.bConfig.2); alarm colour if $typTimetable$.wDayLessonOnce[1].2; toggles $typTimetable$.wDayLessonOnce[1].2
rectangle at (182,110)-(227,136): invisible if NOT $typTimetable$.bConfig.2 AND NOT ($typTimetable$.wDayLessonOnce[1].3 AND NOT $typTimetable$.bConfig.2); alarm colour if $typTimetable$.wDayLessonOnce[1].3; toggles $typTimetable$.wDayLessonOnce[1].3
rectangle at (227,110)-(272,136): invisible if NOT $typTimetable$.bConfig.2 AND NOT ($typTimetable$.wDayLessonOnce[1].4 AND NOT $typTimetable$.bConfig.2); alarm colour if $typTimetable$.wDayLessonOnce[1].4; toggles $typTimetable$.wDayLessonOnce[1].4
rectangle at (272,110)-(317,136): invisible if NOT $typTimetable$.bConfig.2 AND NOT ($typTimetable$.wDayLessonOnce[1].5 AND NOT $typTimetable$.bConfig.2); alarm colour if $typTimetable$.wDayLessonOnce[1].5; toggles $typTimetable$.wDayLessonOnce[1].5
rectangle at (317,110)-(362,136): invisible if NOT $typTimetable$.bConfig.2 AND NOT ($typTimetable$.wDayLessonOnce[1].6 AND NOT $typTimetable$.bConfig.2); alarm colour if $typTimetable$.wDayLessonOnce[1].6; toggles $typTimetable$.wDayLessonOnce[1].6
rectangle at (362,110)-(407,136): invisible if NOT $typTimetable$.bConfig.2 AND NOT ($typTimetable$.wDayLessonOnce[1].7 AND NOT $typTimetable$.bConfig.2); alarm colour if $typTimetable$.wDayLessonOnce[1].7; toggles $typTimetable$.wDayLessonOnce[1].7
rectangle at (407,110)-(452,136): invisible if NOT $typTimetable$.bConfig.2 AND NOT ($typTimetable$.wDayLessonOnce[1].8 AND NOT $typTimetable$.bConfig.2); alarm colour if $typTimetable$.wDayLessonOnce[1].8; toggles $typTimetable$.wDayLessonOnce[1].8
rectangle at (452,110)-(497,136): invisible if NOT $typTimetable$.bConfig.2 AND NOT ($typTimetable$.wDayLessonOnce[1].9 AND NOT $typTimetable$.bConfig.2); alarm colour if $typTimetable$.wDayLessonOnce[1].9; toggles $typTimetable$.wDayLessonOnce[1].9
rectangle at (497,110)-(542,136): invisible if NOT $typTimetable$.bConfig.2 AND NOT ($typTimetable$.wDayLessonOnce[1].10 AND NOT $typTimetable$.bConfig.2); alarm colour if $typTimetable$.wDayLessonOnce[1].10; toggles $typTimetable$.wDayLessonOnce[1].10
rectangle at (542,110)-(587,136): invisible if NOT $typTimetable$.bConfig.2 AND NOT ($typTimetable$.wDayLessonOnce[1].11 AND NOT $typTimetable$.bConfig.2); alarm colour if $typTimetable$.wDayLessonOnce[1].11; toggles $typTimetable$.wDayLessonOnce[1].11
rectangle at (587,110)-(632,136): invisible if NOT $typTimetable$.bConfig.2 AND NOT ($typTimetable$.wDayLessonOnce[1].12 AND NOT $typTimetable$.bConfig.2); alarm colour if $typTimetable$.wDayLessonOnce[1].12; toggles $typTimetable$.wDayLessonOnce[1].12
rectangle at (632,110)-(677,136): invisible if NOT $typTimetable$.bConfig.2 AND NOT ($typTimetable$.wDayLessonOnce[1].13 AND NOT $typTimetable$.bConfig.2); alarm colour if $typTimetable$.wDayLessonOnce[1].13; toggles $typTimetable$.wDayLessonOnce[1].13
rectangle at (677,110)-(722,136): invisible if NOT $typTimetable$.bConfig.2 AND NOT ($typTimetable$.wDayLessonOnce[1].14 AND NOT $typTimetable$.bConfig.2); alarm colour if $typTimetable$.wDayLessonOnce[1].14; toggles $typTimetable$.wDayLessonOnce[1].14
rectangle at (722,110)-(767,136): invisible if NOT $typTimetable$.bConfig.2 AND NOT ($typTimetable$.wDayLessonOnce[1].15 AND NOT $typTimetable$.bConfig.2); alarm colour if $typTimetable$.wDayLessonOnce[1].15; toggles $typTimetable$.wDayLessonOnce[1].15
rectangle at (766,110)-(808,136): invisible if NOT $typTimetable$.bConfig.2 AND NOT ($typTimetable$.wDayLessonOnce[1].0 AND NOT $typTimetable$.bConfig.2); alarm colour if $typTimetable$.wDayLessonOnce[1].0; toggles $typTimetable$.wDayLessonOnce[1].0
rectangle at (92,136)-(137,162): invisible if NOT $typTimetable$.bConfig.2 AND NOT ($typTimetable$.wDayLessonOnce[2].1 AND NOT $typTimetable$.bConfig.2); alarm colour if $typTimetable$.wDayLessonOnce[2].1; toggles $typTimetable$.wDayLessonOnce[2].1
rectangle at (137,136)-(182,162): invisible if NOT $typTimetable$.bConfig.2 AND NOT ($typTimetable$.wDayLessonOnce[2].2 AND NOT $typTimetable$.bConfig.2); alarm colour if $typTimetable$.wDayLessonOnce[2].2; toggles $typTimetable$.wDayLessonOnce[2].2
rectangle at (182,136)-(227,162): invisible if NOT $typTimetable$.bConfig.2 AND NOT ($typTimetable$.wDayLessonOnce[2].3 AND NOT $typTimetable$.bConfig.2); alarm colour if $typTimetable$.wDayLessonOnce[2].3; toggles $typTimetable$.wDayLessonOnce[2].3
rectangle at (227,136)-(272,162): invisible if NOT $typTimetable$.bConfig.2 AND NOT ($typTimetable$.wDayLessonOnce[2].4 AND NOT $typTimetable$.bConfig.2); alarm colour if $typTimetable$.wDayLessonOnce[2].4; toggles $typTimetable$.wDayLessonOnce[2].4
rectangle at (272,136)-(317,162): invisible if NOT $typTimetable$.bConfig.2 AND NOT ($typTimetable$.wDayLessonOnce[2].5 AND NOT $typTimetable$.bConfig.2); alarm colour if $typTimetable$.wDayLessonOnce[2].5; toggles $typTimetable$.wDayLessonOnce[2].5
rectangle at (317,136)-(362,162): invisible if NOT $typTimetable$.bConfig.2 AND NOT ($typTimetable$.wDayLessonOnce[2].6 AND NOT $typTimetable$.bConfig.2); alarm colour if $typTimetable$.wDayLessonOnce[2].6; toggles $typTimetable$.wDayLessonOnce[2].6
rectangle at (362,136)-(407,162): invisible if NOT $typTimetable$.bConfig.2 AND NOT ($typTimetable$.wDayLessonOnce[2].7 AND NOT $typTimetable$.bConfig.2); alarm colour if $typTimetable$.wDayLessonOnce[2].7; toggles $typTimetable$.wDayLessonOnce[2].7
rectangle at (407,136)-(452,162): invisible if NOT $typTimetable$.bConfig.2 AND NOT ($typTimetable$.wDayLessonOnce[2].8 AND NOT $typTimetable$.bConfig.2); alarm colour if $typTimetable$.wDayLessonOnce[2].8; toggles $typTimetable$.wDayLessonOnce[2].8
rectangle at (452,136)-(497,162): invisible if NOT $typTimetable$.bConfig.2 AND NOT ($typTimetable$.wDayLessonOnce[2].9 AND NOT $typTimetable$.bConfig.2); alarm colour if $typTimetable$.wDayLessonOnce[2].9; toggles $typTimetable$.wDayLessonOnce[2].9
rectangle at (497,136)-(542,162): invisible if NOT $typTimetable$.bConfig.2 AND NOT ($typTimetable$.wDayLessonOnce[2].10 AND NOT $typTimetable$.bConfig.2); alarm colour if $typTimetable$.wDayLessonOnce[2].10; toggles $typTimetable$.wDayLessonOnce[2].10
rectangle at (542,136)-(587,162): invisible if NOT $typTimetable$.bConfig.2 AND NOT ($typTimetable$.wDayLessonOnce[2].11 AND NOT $typTimetable$.bConfig.2); alarm colour if $typTimetable$.wDayLessonOnce[2].11; toggles $typTimetable$.wDayLessonOnce[2].11
rectangle at (587,136)-(632,162): invisible if NOT $typTimetable$.bConfig.2 AND NOT ($typTimetable$.wDayLessonOnce[2].12 AND NOT $typTimetable$.bConfig.2); alarm colour if $typTimetable$.wDayLessonOnce[2].12; toggles $typTimetable$.wDayLessonOnce[2].12
rectangle at (632,136)-(677,162): invisible if NOT $typTimetable$.bConfig.2 AND NOT ($typTimetable$.wDayLessonOnce[2].13 AND NOT $typTimetable$.bConfig.2); alarm colour if $typTimetable$.wDayLessonOnce[2].13; toggles $typTimetable$.wDayLessonOnce[2].13
rectangle at (677,136)-(722,162): invisible if NOT $typTimetable$.bConfig.2 AND NOT ($typTimetable$.wDayLessonOnce[2].14 AND NOT $typTimetable$.bConfig.2); alarm colour if $typTimetable$.wDayLessonOnce[2].14; toggles $typTimetable$.wDayLessonOnce[2].14
rectangle at (722,136)-(767,162): invisible if NOT $typTimetable$.bConfig.2 AND NOT ($typTimetable$.wDayLessonOnce[2].15 AND NOT $typTimetable$.bConfig.2); alarm colour if $typTimetable$.wDayLessonOnce[2].15; toggles $typTimetable$.wDayLessonOnce[2].15
rectangle at (766,136)-(808,162): invisible if NOT $typTimetable$.bConfig.2 AND NOT ($typTimetable$.wDayLessonOnce[2].0 AND NOT $typTimetable$.bConfig.2); alarm colour if $typTimetable$.wDayLessonOnce[2].0; toggles $typTimetable$.wDayLessonOnce[2].0
rectangle at (92,162)-(137,188): invisible if NOT $typTimetable$.bConfig.2 AND NOT ($typTimetable$.wDayLessonOnce[3].1 AND NOT $typTimetable$.bConfig.2); alarm colour if $typTimetable$.wDayLessonOnce[3].1; toggles $typTimetable$.wDayLessonOnce[3].1
rectangle at (137,162)-(182,188): invisible if NOT $typTimetable$.bConfig.2 AND NOT ($typTimetable$.wDayLessonOnce[3].2 AND NOT $typTimetable$.bConfig.2); alarm colour if $typTimetable$.wDayLessonOnce[3].2; toggles $typTimetable$.wDayLessonOnce[3].2
rectangle at (182,162)-(227,188): invisible if NOT $typTimetable$.bConfig.2 AND NOT ($typTimetable$.wDayLessonOnce[3].3 AND NOT $typTimetable$.bConfig.2); alarm colour if $typTimetable$.wDayLessonOnce[3].3; toggles $typTimetable$.wDayLessonOnce[3].3
rectangle at (227,162)-(272,188): invisible if NOT $typTimetable$.bConfig.2 AND NOT ($typTimetable$.wDayLessonOnce[3].4 AND NOT $typTimetable$.bConfig.2); alarm colour if $typTimetable$.wDayLessonOnce[3].4; toggles $typTimetable$.wDayLessonOnce[3].4
rectangle at (272,162)-(317,188): invisible if NOT $typTimetable$.bConfig.2 AND NOT ($typTimetable$.wDayLessonOnce[3].5 AND NOT $typTimetable$.bConfig.2); alarm colour if $typTimetable$.wDayLessonOnce[3].5; toggles $typTimetable$.wDayLessonOnce[3].5
rectangle at (317,162)-(362,188): invisible if NOT $typTimetable$.bConfig.2 AND NOT ($typTimetable$.wDayLessonOnce[3].6 AND NOT $typTimetable$.bConfig.2); alarm colour if $typTimetable$.wDayLessonOnce[3].6; toggles $typTimetable$.wDayLessonOnce[3].6
rectangle at (362,162)-(407,188): invisible if NOT $typTimetable$.bConfig.2 AND NOT ($typTimetable$.wDayLessonOnce[3].7 AND NOT $typTimetable$.bConfig.2); alarm colour if $typTimetable$.wDayLessonOnce[3].7; toggles $typTimetable$.wDayLessonOnce[3].7
rectangle at (407,162)-(452,188): invisible if NOT $typTimetable$.bConfig.2 AND NOT ($typTimetable$.wDayLessonOnce[3].8 AND NOT $typTimetable$.bConfig.2); alarm colour if $typTimetable$.wDayLessonOnce[3].8; toggles $typTimetable$.wDayLessonOnce[3].8
rectangle at (452,162)-(497,188): invisible if NOT $typTimetable$.bConfig.2 AND NOT ($typTimetable$.wDayLessonOnce[3].9 AND NOT $typTimetable$.bConfig.2); alarm colour if $typTimetable$.wDayLessonOnce[3].9; toggles $typTimetable$.wDayLessonOnce[3].9
rectangle at (497,162)-(542,188): invisible if NOT $typTimetable$.bConfig.2 AND NOT ($typTimetable$.wDayLessonOnce[3].10 AND NOT $typTimetable$.bConfig.2); alarm colour if $typTimetable$.wDayLessonOnce[3].10; toggles $typTimetable$.wDayLessonOnce[3].10
rectangle at (542,162)-(587,188): invisible if NOT $typTimetable$.bConfig.2 AND NOT ($typTimetable$.wDayLessonOnce[3].11 AND NOT $typTimetable$.bConfig.2); alarm colour if $typTimetable$.wDayLessonOnce[3].11; toggles $typTimetable$.wDayLessonOnce[3].11
rectangle at (587,162)-(632,188): invisible if NOT $typTimetable$.bConfig.2 AND NOT ($typTimetable$.wDayLessonOnce[3].12 AND NOT $typTimetable$.bConfig.2); alarm colour if $typTimetable$.wDayLessonOnce[3].12; toggles $typTimetable$.wDayLessonOnce[3].12
rectangle at (632,162)-(677,188): invisible if NOT $typTimetable$.bConfig.2 AND NOT ($typTimetable$.wDayLessonOnce[3].13 AND NOT $typTimetable$.bConfig.2); alarm colour if $typTimetable$.wDayLessonOnce[3].13; toggles $typTimetable$.wDayLessonOnce[3].13
rectangle at (677,162)-(722,188): invisible if NOT $typTimetable$.bConfig.2 AND NOT ($typTimetable$.wDayLessonOnce[3].14 AND NOT $typTimetable$.bConfig.2); alarm colour if $typTimetable$.wDayLessonOnce[3].14; toggles $typTimetable$.wDayLessonOnce[3].14
rectangle at (722,162)-(767,188): invisible if NOT $typTimetable$.bConfig.2 AND NOT ($typTimetable$.wDayLessonOnce[3].15 AND NOT $typTimetable$.bConfig.2); alarm colour if $typTimetable$.wDayLessonOnce[3].15; toggles $typTimetable$.wDayLessonOnce[3].15
rectangle at (766,162)-(808,188): invisible if NOT $typTimetable$.bConfig.2 AND NOT ($typTimetable$.wDayLessonOnce[3].0 AND NOT $typTimetable$.bConfig.2); alarm colour if $typTimetable$.wDayLessonOnce[3].0; toggles $typTimetable$.wDayLessonOnce[3].0
rectangle at (92,188)-(137,214): invisible if NOT $typTimetable$.bConfig.2 AND NOT ($typTimetable$.wDayLessonOnce[4].1 AND NOT $typTimetable$.bConfig.2); alarm colour if $typTimetable$.wDayLessonOnce[4].1; toggles $typTimetable$.wDayLessonOnce[4].1
rectangle at (137,188)-(182,214): invisible if NOT $typTimetable$.bConfig.2 AND NOT ($typTimetable$.wDayLessonOnce[4].2 AND NOT $typTimetable$.bConfig.2); alarm colour if $typTimetable$.wDayLessonOnce[4].2; toggles $typTimetable$.wDayLessonOnce[4].2
rectangle at (182,188)-(227,214): invisible if NOT $typTimetable$.bConfig.2 AND NOT ($typTimetable$.wDayLessonOnce[4].3 AND NOT $typTimetable$.bConfig.2); alarm colour if $typTimetable$.wDayLessonOnce[4].3; toggles $typTimetable$.wDayLessonOnce[4].3
rectangle at (227,188)-(272,214): invisible if NOT $typTimetable$.bConfig.2 AND NOT ($typTimetable$.wDayLessonOnce[4].4 AND NOT $typTimetable$.bConfig.2); alarm colour if $typTimetable$.wDayLessonOnce[4].4; toggles $typTimetable$.wDayLessonOnce[4].4
rectangle at (272,188)-(317,214): invisible if NOT $typTimetable$.bConfig.2 AND NOT ($typTimetable$.wDayLessonOnce[4].5 AND NOT $typTimetable$.bConfig.2); alarm colour if $typTimetable$.wDayLessonOnce[4].5; toggles $typTimetable$.wDayLessonOnce[4].5
rectangle at (317,188)-(362,214): invisible if NOT $typTimetable$.bConfig.2 AND NOT ($typTimetable$.wDayLessonOnce[4].6 AND NOT $typTimetable$.bConfig.2); alarm colour if $typTimetable$.wDayLessonOnce[4].6; toggles $typTimetable$.wDayLessonOnce[4].6
rectangle at (362,188)-(407,214): invisible if NOT $typTimetable$.bConfig.2 AND NOT ($typTimetable$.wDayLessonOnce[4].7 AND NOT $typTimetable$.bConfig.2); alarm colour if $typTimetable$.wDayLessonOnce[4].7; toggles $typTimetable$.wDayLessonOnce[4].7
rectangle at (407,188)-(452,214): invisible if NOT $typTimetable$.bConfig.2 AND NOT ($typTimetable$.wDayLessonOnce[4].8 AND NOT $typTimetable$.bConfig.2); alarm colour if $typTimetable$.wDayLessonOnce[4].8; toggles $typTimetable$.wDayLessonOnce[4].8
rectangle at (452,188)-(497,214): invisible if NOT $typTimetable$.bConfig.2 AND NOT ($typTimetable$.wDayLessonOnce[4].9 AND NOT $typTimetable$.bConfig.2); alarm colour if $typTimetable$.wDayLessonOnce[4].9; toggles $typTimetable$.wDayLessonOnce[4].9
rectangle at (497,188)-(542,214): invisible if NOT $typTimetable$.bConfig.2 AND NOT ($typTimetable$.wDayLessonOnce[4].10 AND NOT $typTimetable$.bConfig.2); alarm colour if $typTimetable$.wDayLessonOnce[4].10; toggles $typTimetable$.wDayLessonOnce[4].10
rectangle at (542,188)-(587,214): invisible if NOT $typTimetable$.bConfig.2 AND NOT ($typTimetable$.wDayLessonOnce[4].11 AND NOT $typTimetable$.bConfig.2); alarm colour if $typTimetable$.wDayLessonOnce[4].11; toggles $typTimetable$.wDayLessonOnce[4].11
rectangle at (587,188)-(632,214): invisible if NOT $typTimetable$.bConfig.2 AND NOT ($typTimetable$.wDayLessonOnce[4].12 AND NOT $typTimetable$.bConfig.2); alarm colour if $typTimetable$.wDayLessonOnce[4].12; toggles $typTimetable$.wDayLessonOnce[4].12
rectangle at (632,188)-(677,214): invisible if NOT $typTimetable$.bConfig.2 AND NOT ($typTimetable$.wDayLessonOnce[4].13 AND NOT $typTimetable$.bConfig.2); alarm colour if $typTimetable$.wDayLessonOnce[4].13; toggles $typTimetable$.wDayLessonOnce[4].13
rectangle at (677,188)-(722,214): invisible if NOT $typTimetable$.bConfig.2 AND NOT ($typTimetable$.wDayLessonOnce[4].14 AND NOT $typTimetable$.bConfig.2); alarm colour if $typTimetable$.wDayLessonOnce[4].14; toggles $typTimetable$.wDayLessonOnce[4].14
rectangle at (722,188)-(767,214): invisible if NOT $typTimetable$.bConfig.2 AND NOT ($typTimetable$.wDayLessonOnce[4].15 AND NOT $typTimetable$.bConfig.2); alarm colour if $typTimetable$.wDayLessonOnce[4].15; toggles $typTimetable$.wDayLessonOnce[4].15
rectangle at (766,188)-(808,214): invisible if NOT $typTimetable$.bConfig.2 AND NOT ($typTimetable$.wDayLessonOnce[4].0 AND NOT $typTimetable$.bConfig.2); alarm colour if $typTimetable$.wDayLessonOnce[4].0; toggles $typTimetable$.wDayLessonOnce[4].0
rectangle at (92,214)-(137,240): invisible if NOT $typTimetable$.bConfig.2 AND NOT ($typTimetable$.wDayLessonOnce[5].1 AND NOT $typTimetable$.bConfig.2); alarm colour if $typTimetable$.wDayLessonOnce[5].1; toggles $typTimetable$.wDayLessonOnce[5].1
rectangle at (137,214)-(182,240): invisible if NOT $typTimetable$.bConfig.2 AND NOT ($typTimetable$.wDayLessonOnce[5].2 AND NOT $typTimetable$.bConfig.2); alarm colour if $typTimetable$.wDayLessonOnce[5].2; toggles $typTimetable$.wDayLessonOnce[5].2
rectangle at (182,214)-(227,240): invisible if NOT $typTimetable$.bConfig.2 AND NOT ($typTimetable$.wDayLessonOnce[5].3 AND NOT $typTimetable$.bConfig.2); alarm colour if $typTimetable$.wDayLessonOnce[5].3; toggles $typTimetable$.wDayLessonOnce[5].3
rectangle at (227,214)-(272,240): invisible if NOT $typTimetable$.bConfig.2 AND NOT ($typTimetable$.wDayLessonOnce[5].4 AND NOT $typTimetable$.bConfig.2); alarm colour if $typTimetable$.wDayLessonOnce[5].4; toggles $typTimetable$.wDayLessonOnce[5].4
rectangle at (272,214)-(317,240): invisible if NOT $typTimetable$.bConfig.2 AND NOT ($typTimetable$.wDayLessonOnce[5].5 AND NOT $typTimetable$.bConfig.2); alarm colour if $typTimetable$.wDayLessonOnce[5].5; toggles $typTimetable$.wDayLessonOnce[5].5
rectangle at (317,214)-(362,240): invisible if NOT $typTimetable$.bConfig.2 AND NOT ($typTimetable$.wDayLessonOnce[5].6 AND NOT $typTimetable$.bConfig.2); alarm colour if $typTimetable$.wDayLessonOnce[5].6; toggles $typTimetable$.wDayLessonOnce[5].6
rectangle at (362,214)-(407,240): invisible if NOT $typTimetable$.bConfig.2 AND NOT ($typTimetable$.wDayLessonOnce[5].7 AND NOT $typTimetable$.bConfig.2); alarm colour if $typTimetable$.wDayLessonOnce[5].7; toggles $typTimetable$.wDayLessonOnce[5].7
rectangle at (407,214)-(452,240): invisible if NOT $typTimetable$.bConfig.2 AND NOT ($typTimetable$.wDayLessonOnce[5].8 AND NOT $typTimetable$.bConfig.2); alarm colour if $typTimetable$.wDayLessonOnce[5].8; toggles $typTimetable$.wDayLessonOnce[5].8
rectangle at (452,214)-(497,240): invisible if NOT $typTimetable$.bConfig.2 AND NOT ($typTimetable$.wDayLessonOnce[5].9 AND NOT $typTimetable$.bConfig.2); alarm colour if $typTimetable$.wDayLessonOnce[5].9; toggles $typTimetable$.wDayLessonOnce[5].9
rectangle at (497,214)-(542,240): invisible if NOT $typTimetable$.bConfig.2 AND NOT ($typTimetable$.wDayLessonOnce[5].10 AND NOT $typTimetable$.bConfig.2); alarm colour if $typTimetable$.wDayLessonOnce[5].10; toggles $typTimetable$.wDayLessonOnce[5].10
rectangle at (542,214)-(587,240): invisible if NOT $typTimetable$.bConfig.2 AND NOT ($typTimetable$.wDayLessonOnce[5].11 AND NOT $typTimetable$.bConfig.2); alarm colour if $typTimetable$.wDayLessonOnce[5].11; toggles $typTimetable$.wDayLessonOnce[5].11
rectangle at (587,214)-(632,240): invisible if NOT $typTimetable$.bConfig.2 AND NOT ($typTimetable$.wDayLessonOnce[5].12 AND NOT $typTimetable$.bConfig.2); alarm colour if $typTimetable$.wDayLessonOnce[5].12; toggles $typTimetable$.wDayLessonOnce[5].12
rectangle at (632,214)-(677,240): invisible if NOT $typTimetable$.bConfig.2 AND NOT ($typTimetable$.wDayLessonOnce[5].13 AND NOT $typTimetable$.bConfig.2); alarm colour if $typTimetable$.wDayLessonOnce[5].13; toggles $typTimetable$.wDayLessonOnce[5].13
rectangle at (677,214)-(722,240): invisible if NOT $typTimetable$.bConfig.2 AND NOT ($typTimetable$.wDayLessonOnce[5].14 AND NOT $typTimetable$.bConfig.2); alarm colour if $typTimetable$.wDayLessonOnce[5].14; toggles $typTimetable$.wDayLessonOnce[5].14
rectangle at (722,214)-(767,240): invisible if NOT $typTimetable$.bConfig.2 AND NOT ($typTimetable$.wDayLessonOnce[5].15 AND NOT $typTimetable$.bConfig.2); alarm colour if $typTimetable$.wDayLessonOnce[5].15; toggles $typTimetable$.wDayLessonOnce[5].15
rectangle at (766,214)-(808,240): invisible if NOT $typTimetable$.bConfig.2 AND NOT ($typTimetable$.wDayLessonOnce[5].0 AND NOT $typTimetable$.bConfig.2); alarm colour if $typTimetable$.wDayLessonOnce[5].0; toggles $typTimetable$.wDayLessonOnce[5].0
rectangle at (92,350)-(137,376): invisible if NOT $typTimetable$.bConfig.2 AND NOT ($typTimetable$.wDayLessonOnce[6].1 AND NOT $typTimetable$.bConfig.2); alarm colour if $typTimetable$.wDayLessonOnce[6].1; toggles $typTimetable$.wDayLessonOnce[6].1
rectangle at (137,350)-(182,376): invisible if NOT $typTimetable$.bConfig.2 AND NOT ($typTimetable$.wDayLessonOnce[6].2 AND NOT $typTimetable$.bConfig.2); alarm colour if $typTimetable$.wDayLessonOnce[6].2; toggles $typTimetable$.wDayLessonOnce[6].2
rectangle at (182,350)-(227,376): invisible if NOT $typTimetable$.bConfig.2 AND NOT ($typTimetable$.wDayLessonOnce[6].3 AND NOT $typTimetable$.bConfig.2); alarm colour if $typTimetable$.wDayLessonOnce[6].3; toggles $typTimetable$.wDayLessonOnce[6].3
rectangle at (227,350)-(272,376): invisible if NOT $typTimetable$.bConfig.2 AND NOT ($typTimetable$.wDayLessonOnce[6].4 AND NOT $typTimetable$.bConfig.2); alarm colour if $typTimetable$.wDayLessonOnce[6].4; toggles $typTimetable$.wDayLessonOnce[6].4
rectangle at (272,350)-(317,376): invisible if NOT $typTimetable$.bConfig.2 AND NOT ($typTimetable$.wDayLessonOnce[6].5 AND NOT $typTimetable$.bConfig.2); alarm colour if $typTimetable$.wDayLessonOnce[6].5; toggles $typTimetable$.wDayLessonOnce[6].5
rectangle at (317,350)-(362,376): invisible if NOT $typTimetable$.bConfig.2 AND NOT ($typTimetable$.wDayLessonOnce[6].6 AND NOT $typTimetable$.bConfig.2); alarm colour if $typTimetable$.wDayLessonOnce[6].6; toggles $typTimetable$.wDayLessonOnce[6].6
rectangle at (362,350)-(407,376): invisible if NOT $typTimetable$.bConfig.2 AND NOT ($typTimetable$.wDayLessonOnce[6].7 AND NOT $typTimetable$.bConfig.2); alarm colour if $typTimetable$.wDayLessonOnce[6].7; toggles $typTimetable$.wDayLessonOnce[6].7
rectangle at (407,350)-(452,376): invisible if NOT $typTimetable$.bConfig.2 AND NOT ($typTimetable$.wDayLessonOnce[6].8 AND NOT $typTimetable$.bConfig.2); alarm colour if $typTimetable$.wDayLessonOnce[6].8; toggles $typTimetable$.wDayLessonOnce[6].8
rectangle at (452,350)-(497,376): invisible if NOT $typTimetable$.bConfig.2 AND NOT ($typTimetable$.wDayLessonOnce[6].9 AND NOT $typTimetable$.bConfig.2); alarm colour if $typTimetable$.wDayLessonOnce[6].9; toggles $typTimetable$.wDayLessonOnce[6].9
rectangle at (497,350)-(542,376): invisible if NOT $typTimetable$.bConfig.2 AND NOT ($typTimetable$.wDayLessonOnce[6].10 AND NOT $typTimetable$.bConfig.2); alarm colour if $typTimetable$.wDayLessonOnce[6].10; toggles $typTimetable$.wDayLessonOnce[6].10
rectangle at (542,350)-(587,376): invisible if NOT $typTimetable$.bConfig.2 AND NOT ($typTimetable$.wDayLessonOnce[6].11 AND NOT $typTimetable$.bConfig.2); alarm colour if $typTimetable$.wDayLessonOnce[6].11; toggles $typTimetable$.wDayLessonOnce[6].11
rectangle at (587,350)-(632,376): invisible if NOT $typTimetable$.bConfig.2 AND NOT ($typTimetable$.wDayLessonOnce[6].12 AND NOT $typTimetable$.bConfig.2); alarm colour if $typTimetable$.wDayLessonOnce[6].12; toggles $typTimetable$.wDayLessonOnce[6].12
rectangle at (632,350)-(677,376): invisible if NOT $typTimetable$.bConfig.2 AND NOT ($typTimetable$.wDayLessonOnce[6].13 AND NOT $typTimetable$.bConfig.2); alarm colour if $typTimetable$.wDayLessonOnce[6].13; toggles $typTimetable$.wDayLessonOnce[6].13
rectangle at (677,350)-(722,376): invisible if NOT $typTimetable$.bConfig.2 AND NOT ($typTimetable$.wDayLessonOnce[6].14 AND NOT $typTimetable$.bConfig.2); alarm colour if $typTimetable$.wDayLessonOnce[6].14; toggles $typTimetable$.wDayLessonOnce[6].14
rectangle at (722,350)-(767,376): invisible if NOT $typTimetable$.bConfig.2 AND NOT ($typTimetable$.wDayLessonOnce[6].15 AND NOT $typTimetable$.bConfig.2); alarm colour if $typTimetable$.wDayLessonOnce[6].15; toggles $typTimetable$.wDayLessonOnce[6].15
rectangle at (766,350)-(808,376): invisible if NOT $typTimetable$.bConfig.2 AND NOT ($typTimetable$.wDayLessonOnce[6].0 AND NOT $typTimetable$.bConfig.2); alarm colour if $typTimetable$.wDayLessonOnce[6].0; toggles $typTimetable$.wDayLessonOnce[6].0
rectangle at (92,376)-(137,402): invisible if NOT $typTimetable$.bConfig.2 AND NOT ($typTimetable$.wDayLessonOnce[7].1 AND NOT $typTimetable$.bConfig.2); alarm colour if $typTimetable$.wDayLessonOnce[7].1; toggles $typTimetable$.wDayLessonOnce[7].1
rectangle at (137,376)-(182,402): invisible if NOT $typTimetable$.bConfig.2 AND NOT ($typTimetable$.wDayLessonOnce[7].2 AND NOT $typTimetable$.bConfig.2); alarm colour if $typTimetable$.wDayLessonOnce[7].2; toggles $typTimetable$.wDayLessonOnce[7].2
rectangle at (182,376)-(227,402): invisible if NOT $typTimetable$.bConfig.2 AND NOT ($typTimetable$.wDayLessonOnce[7].3 AND NOT $typTimetable$.bConfig.2); alarm colour if $typTimetable$.wDayLessonOnce[7].3; toggles $typTimetable$.wDayLessonOnce[6].3
rectangle at (227,376)-(272,402): invisible if NOT $typTimetable$.bConfig.2 AND NOT ($typTimetable$.wDayLessonOnce[7].4 AND NOT $typTimetable$.bConfig.2); alarm colour if $typTimetable$.wDayLessonOnce[7].4; toggles $typTimetable$.wDayLessonOnce[7].4
rectangle at (272,376)-(317,402): invisible if NOT $typTimetable$.bConfig.2 AND NOT ($typTimetable$.wDayLessonOnce[7].5 AND NOT $typTimetable$.bConfig.2); alarm colour if $typTimetable$.wDayLessonOnce[7].5; toggles $typTimetable$.wDayLessonOnce[7].5
rectangle at (317,376)-(362,402): invisible if NOT $typTimetable$.bConfig.2 AND NOT ($typTimetable$.wDayLessonOnce[7].6 AND NOT $typTimetable$.bConfig.2); alarm colour if $typTimetable$.wDayLessonOnce[7].6; toggles $typTimetable$.wDayLessonOnce[7].6
rectangle at (362,376)-(407,402): invisible if NOT $typTimetable$.bConfig.2 AND NOT ($typTimetable$.wDayLessonOnce[7].7 AND NOT $typTimetable$.bConfig.2); alarm colour if $typTimetable$.wDayLessonOnce[7].7; toggles $typTimetable$.wDayLessonOnce[7].7
rectangle at (407,376)-(452,402): invisible if NOT $typTimetable$.bConfig.2 AND NOT ($typTimetable$.wDayLessonOnce[7].8 AND NOT $typTimetable$.bConfig.2); alarm colour if $typTimetable$.wDayLessonOnce[7].8; toggles $typTimetable$.wDayLessonOnce[7].8
rectangle at (452,376)-(497,402): invisible if NOT $typTimetable$.bConfig.2 AND NOT ($typTimetable$.wDayLessonOnce[7].9 AND NOT $typTimetable$.bConfig.2); alarm colour if $typTimetable$.wDayLessonOnce[7].9; toggles $typTimetable$.wDayLessonOnce[7].9
rectangle at (497,376)-(542,402): invisible if NOT $typTimetable$.bConfig.2 AND NOT ($typTimetable$.wDayLessonOnce[7].10 AND NOT $typTimetable$.bConfig.2); alarm colour if $typTimetable$.wDayLessonOnce[7].10; toggles $typTimetable$.wDayLessonOnce[7].10
rectangle at (542,376)-(587,402): invisible if NOT $typTimetable$.bConfig.2 AND NOT ($typTimetable$.wDayLessonOnce[7].11 AND NOT $typTimetable$.bConfig.2); alarm colour if $typTimetable$.wDayLessonOnce[7].11; toggles $typTimetable$.wDayLessonOnce[7].11
rectangle at (587,376)-(632,402): invisible if NOT $typTimetable$.bConfig.2 AND NOT ($typTimetable$.wDayLessonOnce[7].12 AND NOT $typTimetable$.bConfig.2); alarm colour if $typTimetable$.wDayLessonOnce[7].12; toggles $typTimetable$.wDayLessonOnce[7].12
rectangle at (632,376)-(677,402): invisible if NOT $typTimetable$.bConfig.2 AND NOT ($typTimetable$.wDayLessonOnce[7].13 AND NOT $typTimetable$.bConfig.2); alarm colour if $typTimetable$.wDayLessonOnce[7].13; toggles $typTimetable$.wDayLessonOnce[7].13
rectangle at (677,376)-(722,402): invisible if NOT $typTimetable$.bConfig.2 AND NOT ($typTimetable$.wDayLessonOnce[7].14 AND NOT $typTimetable$.bConfig.2); alarm colour if $typTimetable$.wDayLessonOnce[7].14; toggles $typTimetable$.wDayLessonOnce[7].14
rectangle at (722,376)-(767,402): invisible if NOT $typTimetable$.bConfig.2 AND NOT ($typTimetable$.wDayLessonOnce[7].15 AND NOT $typTimetable$.bConfig.2); alarm colour if $typTimetable$.wDayLessonOnce[7].15; toggles $typTimetable$.wDayLessonOnce[7].15
rectangle at (766,376)-(808,402): invisible if NOT $typTimetable$.bConfig.2 AND NOT ($typTimetable$.wDayLessonOnce[7].0 AND NOT $typTimetable$.bConfig.2); alarm colour if $typTimetable$.wDayLessonOnce[7].0; toggles $typTimetable$.wDayLessonOnce[7].0
rectangle at (190,414)-(287,442): text "once run"
rectangle at (855,214)-(900,240): text ":"; tooltip Switch ON time of the scheduler single weekly
rectangle at (264,419)-(281,436): toggles $typTimetable$.bConfig.2; tooltip selection once run enable/disable
polyline at (265,420)-(278,434): invisible if NOT $typTimetable$.bConfig.2; toggles $typTimetable$.bConfig.2
rectangle at (491,452)-(520,477): invisible if $typTimetable$.bStatus.0 OR $typTimetable$.bStatus.1
rectangle at (491,452)-(520,477): invisible if $typTimetable$.bStatus.0 OR $typTimetable$.bStatus.1 OR $typTimetable$.bStatus.3
rectangle at (860,219)-(875,235): text "%0.2d"; shows $typTimetable$.wEveningOff_hour[5]; editable 0..23
rectangle at (880,219)-(895,235): text "%0.2d"; shows $typTimetable$.wEveningOff_minute[5]; editable 0..59
6 more shapes without text or variables
*)

(* Visualisation visuTimetable_Lesson
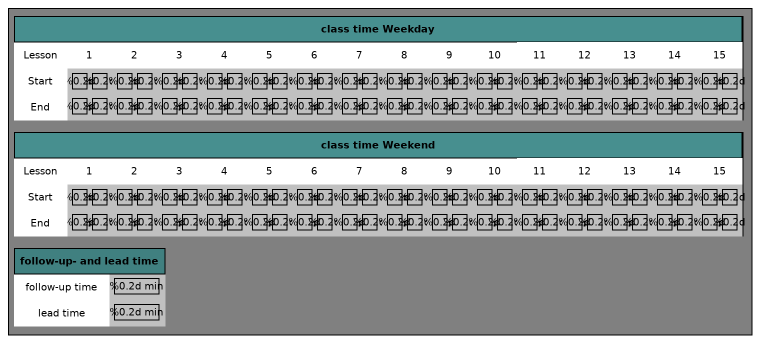
rectangle at (59,60)-(104,86): text ":"; tooltip Switch ON time
rectangle at (64,65)-(79,81): text "%0.2d"; shows $typLesson$.wWeekdayOn_hour[1]; editable 0..23
rectangle at (84,65)-(99,81): text "%0.2d"; shows $typLesson$.wWeekdayOn_Minute[1]; editable 0..59
rectangle at (59,86)-(104,112): text ":"; tooltip Switch OFF time
rectangle at (64,90)-(79,106): text "%0.2d"; shows $typLesson$.wWeekdayOff_hour[1]; editable 0..23
rectangle at (84,90)-(99,106): text "%0.2d"; shows $typLesson$.wWeekdayOff_Minute[1]; editable 0..59
rectangle at (104,60)-(149,86): text ":"; tooltip Switch ON time
rectangle at (109,65)-(124,81): text "%0.2d"; shows $typLesson$.wWeekdayOn_hour[2]; editable 0..23
rectangle at (129,65)-(144,81): text "%0.2d"; shows $typLesson$.wWeekdayOn_Minute[2]; editable 0..59
rectangle at (104,86)-(149,112): text ":"; tooltip Switch OFF time
rectangle at (109,90)-(124,106): text "%0.2d"; shows $typLesson$.wWeekdayOff_hour[2]; editable 0..23
rectangle at (129,90)-(144,106): text "%0.2d"; shows $typLesson$.wWeekdayOff_Minute[2]; editable 0..59
rectangle at (149,60)-(194,86): text ":"; tooltip Switch ON time
rectangle at (154,65)-(169,81): text "%0.2d"; shows $typLesson$.wWeekdayOn_hour[3]; editable 0..23
rectangle at (174,65)-(189,81): text "%0.2d"; shows $typLesson$.wWeekdayOn_Minute[3]; editable 0..59
rectangle at (149,86)-(194,112): text ":"; tooltip Switch OFF time
rectangle at (154,90)-(169,106): text "%0.2d"; shows $typLesson$.wWeekdayOff_hour[3]; editable 0..23
rectangle at (174,90)-(189,106): text "%0.2d"; shows $typLesson$.wWeekdayOff_Minute[3]; editable 0..59
rectangle at (194,60)-(239,86): text ":"; tooltip Switch ON time
rectangle at (199,65)-(214,81): text "%0.2d"; shows $typLesson$.wWeekdayOn_hour[4]; editable 0..23
rectangle at (219,65)-(234,81): text "%0.2d"; shows $typLesson$.wWeekdayOn_Minute[4]; editable 0..59
rectangle at (194,86)-(239,112): text ":"; tooltip Switch OFF time
rectangle at (199,90)-(214,106): text "%0.2d"; shows $typLesson$.wWeekdayOff_hour[4]; editable 0..23
rectangle at (219,90)-(234,106): text "%0.2d"; shows $typLesson$.wWeekdayOff_Minute[4]; editable 0..59
rectangle at (239,60)-(284,86): text ":"; tooltip Switch ON time
rectangle at (244,65)-(259,81): text "%0.2d"; shows $typLesson$.wWeekdayOn_hour[5]; editable 0..23
rectangle at (264,65)-(279,81): text "%0.2d"; shows $typLesson$.wWeekdayOn_Minute[5]; editable 0..59
rectangle at (239,86)-(284,112): text ":"; tooltip Switch OFF time
rectangle at (244,90)-(259,106): text "%0.2d"; shows $typLesson$.wWeekdayOff_hour[5]; editable 0..23
rectangle at (264,90)-(279,106): text "%0.2d"; shows $typLesson$.wWeekdayOff_Minute[5]; editable 0..59
rectangle at (284,60)-(329,86): text ":"; tooltip Switch ON time
rectangle at (289,65)-(304,81): text "%0.2d"; shows $typLesson$.wWeekdayOn_hour[6]; editable 0..23
rectangle at (309,65)-(324,81): text "%0.2d"; shows $typLesson$.wWeekdayOn_Minute[6]; editable 0..59
rectangle at (284,86)-(329,112): text ":"; tooltip Switch OFF time
rectangle at (289,90)-(304,106): text "%0.2d"; shows $typLesson$.wWeekdayOff_hour[6]; editable 0..23
rectangle at (309,90)-(324,106): text "%0.2d"; shows $typLesson$.wWeekdayOff_Minute[6]; editable 0..59
rectangle at (329,60)-(374,86): text ":"; tooltip Switch ON time
rectangle at (334,65)-(349,81): text "%0.2d"; shows $typLesson$.wWeekdayOn_hour[7]; editable 0..23
rectangle at (354,65)-(369,81): text "%0.2d"; shows $typLesson$.wWeekdayOn_Minute[7]; editable 0..59
rectangle at (329,86)-(374,112): text ":"; tooltip Switch OFF time
rectangle at (334,90)-(349,106): text "%0.2d"; shows $typLesson$.wWeekdayOff_hour[7]; editable 0..23
rectangle at (354,90)-(369,106): text "%0.2d"; shows $typLesson$.wWeekdayOff_Minute[7]; editable 0..59
rectangle at (374,60)-(419,86): text ":"; tooltip Switch ON time
rectangle at (379,65)-(394,81): text "%0.2d"; shows $typLesson$.wWeekdayOn_hour[8]; editable 0..23
rectangle at (399,65)-(414,81): text "%0.2d"; shows $typLesson$.wWeekdayOn_Minute[8]; editable 0..59
rectangle at (374,86)-(419,112): text ":"; tooltip Switch OFF time
rectangle at (379,90)-(394,106): text "%0.2d"; shows $typLesson$.wWeekdayOff_hour[8]; editable 0..23
rectangle at (399,90)-(414,106): text "%0.2d"; shows $typLesson$.wWeekdayOff_Minute[8]; editable 0..59
rectangle at (419,60)-(464,86): text ":"; tooltip Switch ON time
rectangle at (424,65)-(439,81): text "%0.2d"; shows $typLesson$.wWeekdayOn_hour[9]; editable 0..23
rectangle at (444,65)-(459,81): text "%0.2d"; shows $typLesson$.wWeekdayOn_Minute[9]; editable 0..59
rectangle at (419,86)-(464,112): text ":"; tooltip Switch OFF time
rectangle at (424,90)-(439,106): text "%0.2d"; shows $typLesson$.wWeekdayOff_hour[9]; editable 0..23
rectangle at (444,90)-(459,106): text "%0.2d"; shows $typLesson$.wWeekdayOff_Minute[9]; editable 0..59
rectangle at (464,60)-(509,86): text ":"; tooltip Switch ON time
rectangle at (469,65)-(484,81): text "%0.2d"; shows $typLesson$.wWeekdayOn_hour[10]; editable 0..23
rectangle at (489,65)-(504,81): text "%0.2d"; shows $typLesson$.wWeekdayOn_Minute[10]; editable 0..59
rectangle at (464,86)-(509,112): text ":"; tooltip Switch OFF time
rectangle at (469,90)-(484,106): text "%0.2d"; shows $typLesson$.wWeekdayOff_hour[10]; editable 0..23
rectangle at (489,90)-(504,106): text "%0.2d"; shows $typLesson$.wWeekdayOff_Minute[10]; editable 0..59
rectangle at (6,60)-(59,86): text "Start"
rectangle at (6,86)-(59,112): text "End"
rectangle at (6,34)-(59,60): text "Lesson"
rectangle at (59,34)-(104,60): text "1"
rectangle at (104,34)-(149,60): text "2"
rectangle at (149,34)-(194,60): text "3"
rectangle at (194,34)-(239,60): text "4"
rectangle at (239,34)-(284,60): text "5"
rectangle at (284,34)-(329,60): text "6"
rectangle at (329,34)-(374,60): text "7"
rectangle at (374,34)-(419,60): text "8"
rectangle at (419,34)-(464,60): text "9"
rectangle at (464,34)-(509,60): text "10"
rectangle at (6,8)-(734,34): text "class time Weekday"
rectangle at (59,176)-(104,202): text ":"; tooltip Switch ON time
rectangle at (64,181)-(79,197): text "%0.2d"; shows $typLesson$.wWeekendOn_hour[1]; editable 0..23
rectangle at (84,181)-(99,197): text "%0.2d"; shows $typLesson$.wWeekendOn_Minute[1]; editable 0..59
rectangle at (59,202)-(104,228): text ":"; tooltip Switch OFF time
rectangle at (64,206)-(79,222): text "%0.2d"; shows $typLesson$.wWeekendOff_hour[1]; editable 0..23
rectangle at (84,206)-(99,222): text "%0.2d"; shows $typLesson$.wWeekendOff_Minute[1]; editable 0..59
rectangle at (104,176)-(149,202): text ":"; tooltip Switch ON time
rectangle at (109,181)-(124,197): text "%0.2d"; shows $typLesson$.wWeekendOn_hour[2]; editable 0..23
rectangle at (129,181)-(144,197): text "%0.2d"; shows $typLesson$.wWeekendOn_Minute[2]; editable 0..59
rectangle at (104,202)-(149,228): text ":"; tooltip Switch OFF time
rectangle at (109,206)-(124,222): text "%0.2d"; shows $typLesson$.wWeekendOff_hour[2]; editable 0..23
rectangle at (129,206)-(144,222): text "%0.2d"; shows $typLesson$.wWeekendOff_Minute[2]; editable 0..59
rectangle at (149,176)-(194,202): text ":"; tooltip Switch ON time
rectangle at (154,181)-(169,197): text "%0.2d"; shows $typLesson$.wWeekendOn_hour[3]; editable 0..23
rectangle at (174,181)-(189,197): text "%0.2d"; shows $typLesson$.wWeekendOn_Minute[3]; editable 0..59
rectangle at (149,202)-(194,228): text ":"; tooltip Switch OFF time
rectangle at (154,206)-(169,222): text "%0.2d"; shows $typLesson$.wWeekendOff_hour[3]; editable 0..23
rectangle at (174,206)-(189,222): text "%0.2d"; shows $typLesson$.wWeekendOff_Minute[3]; editable 0..59
rectangle at (194,176)-(239,202): text ":"; tooltip Switch ON time
rectangle at (199,181)-(214,197): text "%0.2d"; shows $typLesson$.wWeekendOn_hour[4]; editable 0..23
rectangle at (219,181)-(234,197): text "%0.2d"; shows $typLesson$.wWeekendOn_Minute[4]; editable 0..59
rectangle at (194,202)-(239,228): text ":"; tooltip Switch OFF time
rectangle at (199,206)-(214,222): text "%0.2d"; shows $typLesson$.wWeekendOff_hour[4]; editable 0..23
rectangle at (219,206)-(234,222): text "%0.2d"; shows $typLesson$.wWeekendOff_Minute[4]; editable 0..59
rectangle at (239,176)-(284,202): text ":"; tooltip Switch ON time
rectangle at (244,181)-(259,197): text "%0.2d"; shows $typLesson$.wWeekendOn_hour[5]; editable 0..23
rectangle at (264,181)-(279,197): text "%0.2d"; shows $typLesson$.wWeekendOn_Minute[5]; editable 0..59
rectangle at (239,202)-(284,228): text ":"; tooltip Switch OFF time
rectangle at (244,206)-(259,222): text "%0.2d"; shows $typLesson$.wWeekendOff_hour[5]; editable 0..23
rectangle at (264,206)-(279,222): text "%0.2d"; shows $typLesson$.wWeekendOff_Minute[5]; editable 0..59
rectangle at (284,176)-(329,202): text ":"; tooltip Switch ON time
rectangle at (289,181)-(304,197): text "%0.2d"; shows $typLesson$.wWeekendOn_hour[6]; editable 0..23
rectangle at (309,181)-(324,197): text "%0.2d"; shows $typLesson$.wWeekendOn_Minute[6]; editable 0..59
rectangle at (284,202)-(329,228): text ":"; tooltip Switch OFF time
rectangle at (289,206)-(304,222): text "%0.2d"; shows $typLesson$.wWeekendOff_hour[6]; editable 0..23
rectangle at (309,206)-(324,222): text "%0.2d"; shows $typLesson$.wWeekendOff_Minute[6]; editable 0..59
rectangle at (329,176)-(374,202): text ":"; tooltip Switch ON time
rectangle at (334,181)-(349,197): text "%0.2d"; shows $typLesson$.wWeekendOn_hour[7]; editable 0..23
rectangle at (354,181)-(369,197): text "%0.2d"; shows $typLesson$.wWeekendOn_Minute[7]; editable 0..59
rectangle at (329,202)-(374,228): text ":"; tooltip Switch OFF time
rectangle at (334,206)-(349,222): text "%0.2d"; shows $typLesson$.wWeekendOff_hour[7]; editable 0..23
rectangle at (354,206)-(369,222): text "%0.2d"; shows $typLesson$.wWeekendOff_Minute[7]; editable 0..59
rectangle at (374,176)-(419,202): text ":"; tooltip Switch ON time
rectangle at (379,181)-(394,197): text "%0.2d"; shows $typLesson$.wWeekendOn_hour[8]; editable 0..23
rectangle at (399,181)-(414,197): text "%0.2d"; shows $typLesson$.wWeekendOn_Minute[8]; editable 0..59
rectangle at (374,202)-(419,228): text ":"; tooltip Switch OFF time
rectangle at (379,206)-(394,222): text "%0.2d"; shows $typLesson$.wWeekendOff_hour[8]; editable 0..23
rectangle at (399,206)-(414,222): text "%0.2d"; shows $typLesson$.wWeekendOff_Minute[8]; editable 0..59
rectangle at (419,176)-(464,202): text ":"; tooltip Switch ON time
rectangle at (424,181)-(439,197): text "%0.2d"; shows $typLesson$.wWeekendOn_hour[9]; editable 0..23
rectangle at (444,181)-(459,197): text "%0.2d"; shows $typLesson$.wWeekendOn_Minute[9]; editable 0..59
rectangle at (419,202)-(464,228): text ":"; tooltip Switch OFF time
rectangle at (424,206)-(439,222): text "%0.2d"; shows $typLesson$.wWeekendOff_hour[9]; editable 0..23
rectangle at (444,206)-(459,222): text "%0.2d"; shows $typLesson$.wWeekendOff_Minute[9]; editable 0..59
rectangle at (464,176)-(509,202): text ":"; tooltip Switch ON time
rectangle at (469,181)-(484,197): text "%0.2d"; shows $typLesson$.wWeekendOn_hour[10]; editable 0..23
rectangle at (489,181)-(504,197): text "%0.2d"; shows $typLesson$.wWeekendOn_Minute[10]; editable 0..59
rectangle at (464,202)-(509,228): text ":"; tooltip Switch OFF time
rectangle at (469,206)-(484,222): text "%0.2d"; shows $typLesson$.wWeekendOff_hour[10]; editable 0..23
rectangle at (489,206)-(504,222): text "%0.2d"; shows $typLesson$.wWeekendOff_Minute[10]; editable 0..59
rectangle at (6,176)-(59,202): text "Start"
rectangle at (6,202)-(59,228): text "End"
rectangle at (6,150)-(59,176): text "Lesson"
rectangle at (59,150)-(104,176): text "1"
rectangle at (104,150)-(149,176): text "2"
rectangle at (149,150)-(194,176): text "3"
rectangle at (194,150)-(239,176): text "4"
rectangle at (239,150)-(284,176): text "5"
rectangle at (284,150)-(329,176): text "6"
rectangle at (329,150)-(374,176): text "7"
rectangle at (374,150)-(419,176): text "8"
rectangle at (419,150)-(464,176): text "9"
rectangle at (464,150)-(509,176): text "10"
rectangle at (6,124)-(734,150): text "class time Weekend"
rectangle at (101,292)-(157,318): tooltip Switch OFF time
rectangle at (106,296)-(151,312): text "%0.2d min"; shows $typLesson$.wLeadTime; editable 0..99
rectangle at (6,292)-(101,318): text "lead time"
rectangle at (101,266)-(157,292): tooltip Switch ON time
rectangle at (106,270)-(151,286): text "%0.2d min"; shows $typLesson$.wFollowupTime; editable 0..99
rectangle at (6,266)-(101,292): text "follow-up time"
rectangle at (6,240)-(157,266): text "follow-up- and lead time"
rectangle at (509,60)-(554,86): text ":"; tooltip Switch ON time
rectangle at (514,65)-(529,81): text "%0.2d"; shows $typLesson$.wWeekdayOn_hour[11]; editable 0..23
rectangle at (534,65)-(549,81): text "%0.2d"; shows $typLesson$.wWeekdayOn_Minute[11]; editable 0..59
rectangle at (509,86)-(554,112): text ":"; tooltip Switch OFF time
rectangle at (514,90)-(529,106): text "%0.2d"; shows $typLesson$.wWeekdayOff_hour[11]; editable 0..23
rectangle at (534,90)-(549,106): text "%0.2d"; shows $typLesson$.wWeekdayOff_Minute[11]; editable 0..59
rectangle at (509,34)-(554,60): text "11"
rectangle at (509,176)-(554,202): text ":"; tooltip Switch ON time
rectangle at (514,181)-(529,197): text "%0.2d"; shows $typLesson$.wWeekendOn_hour[11]; editable 0..23
rectangle at (534,181)-(549,197): text "%0.2d"; shows $typLesson$.wWeekendOn_Minute[11]; editable 0..59
rectangle at (509,202)-(554,228): text ":"; tooltip Switch OFF time
rectangle at (514,206)-(529,222): text "%0.2d"; shows $typLesson$.wWeekendOff_hour[11]; editable 0..23
rectangle at (534,206)-(549,222): text "%0.2d"; shows $typLesson$.wWeekendOff_Minute[11]; editable 0..59
rectangle at (509,150)-(554,176): text "11"
rectangle at (554,60)-(599,86): text ":"; tooltip Switch ON time
rectangle at (559,65)-(574,81): text "%0.2d"; shows $typLesson$.wWeekdayOn_hour[12]; editable 0..23
rectangle at (579,65)-(594,81): text "%0.2d"; shows $typLesson$.wWeekdayOn_Minute[12]; editable 0..59
rectangle at (554,86)-(599,112): text ":"; tooltip Switch OFF time
rectangle at (559,90)-(574,106): text "%0.2d"; shows $typLesson$.wWeekdayOff_hour[12]; editable 0..23
rectangle at (579,90)-(594,106): text "%0.2d"; shows $typLesson$.wWeekdayOff_Minute[12]; editable 0..59
rectangle at (554,34)-(599,60): text "12"
rectangle at (554,176)-(599,202): text ":"; tooltip Switch ON time
rectangle at (559,181)-(574,197): text "%0.2d"; shows $typLesson$.wWeekendOn_hour[12]; editable 0..23
rectangle at (579,181)-(594,197): text "%0.2d"; shows $typLesson$.wWeekendOn_Minute[12]; editable 0..59
rectangle at (554,202)-(599,228): text ":"; tooltip Switch OFF time
rectangle at (559,206)-(574,222): text "%0.2d"; shows $typLesson$.wWeekendOff_hour[12]; editable 0..23
rectangle at (579,206)-(594,222): text "%0.2d"; shows $typLesson$.wWeekendOff_Minute[12]; editable 0..59
rectangle at (554,150)-(599,176): text "12"
rectangle at (599,60)-(644,86): text ":"; tooltip Switch ON time
rectangle at (604,65)-(619,81): text "%0.2d"; shows $typLesson$.wWeekdayOn_hour[13]; editable 0..23
rectangle at (624,65)-(639,81): text "%0.2d"; shows $typLesson$.wWeekdayOn_Minute[13]; editable 0..59
rectangle at (599,86)-(644,112): text ":"; tooltip Switch OFF time
rectangle at (604,90)-(619,106): text "%0.2d"; shows $typLesson$.wWeekdayOff_hour[13]; editable 0..23
rectangle at (624,90)-(639,106): text "%0.2d"; shows $typLesson$.wWeekdayOff_Minute[13]; editable 0..59
rectangle at (599,34)-(644,60): text "13"
rectangle at (599,176)-(644,202): text ":"; tooltip Switch ON time
rectangle at (604,181)-(619,197): text "%0.2d"; shows $typLesson$.wWeekendOn_hour[13]; editable 0..23
rectangle at (624,181)-(639,197): text "%0.2d"; shows $typLesson$.wWeekendOn_Minute[13]; editable 0..59
rectangle at (599,202)-(644,228): text ":"; tooltip Switch OFF time
rectangle at (604,206)-(619,222): text "%0.2d"; shows $typLesson$.wWeekendOff_hour[13]; editable 0..23
rectangle at (624,206)-(639,222): text "%0.2d"; shows $typLesson$.wWeekendOff_Minute[13]; editable 0..59
rectangle at (599,150)-(644,176): text "13"
rectangle at (644,60)-(689,86): text ":"; tooltip Switch ON time
rectangle at (649,65)-(664,81): text "%0.2d"; shows $typLesson$.wWeekdayOn_hour[14]; editable 0..23
rectangle at (669,65)-(684,81): text "%0.2d"; shows $typLesson$.wWeekdayOn_Minute[14]; editable 0..59
rectangle at (644,86)-(689,112): text ":"; tooltip Switch OFF time
rectangle at (649,90)-(664,106): text "%0.2d"; shows $typLesson$.wWeekdayOff_hour[14]; editable 0..23
rectangle at (669,90)-(684,106): text "%0.2d"; shows $typLesson$.wWeekdayOff_Minute[14]; editable 0..59
rectangle at (644,34)-(689,60): text "14"
rectangle at (644,176)-(689,202): text ":"; tooltip Switch ON time
rectangle at (649,181)-(664,197): text "%0.2d"; shows $typLesson$.wWeekendOn_hour[14]; editable 0..23
rectangle at (669,181)-(684,197): text "%0.2d"; shows $typLesson$.wWeekendOn_Minute[14]; editable 0..59
rectangle at (644,202)-(689,228): text ":"; tooltip Switch OFF time
rectangle at (649,206)-(664,222): text "%0.2d"; shows $typLesson$.wWeekendOff_hour[14]; editable 0..23
rectangle at (669,206)-(684,222): text "%0.2d"; shows $typLesson$.wWeekendOff_Minute[14]; editable 0..59
rectangle at (644,150)-(689,176): text "14"
rectangle at (689,60)-(734,86): text ":"; tooltip Switch ON time
rectangle at (694,65)-(709,81): text "%0.2d"; shows $typLesson$.wWeekdayOn_hour[15]; editable 0..23
rectangle at (714,65)-(729,81): text "%0.2d"; shows $typLesson$.wWeekdayOn_Minute[15]; editable 0..59
rectangle at (689,86)-(734,112): text ":"; tooltip Switch OFF time
rectangle at (694,90)-(709,106): text "%0.2d"; shows $typLesson$.wWeekdayOff_hour[15]; editable 0..23
rectangle at (714,90)-(729,106): text "%0.2d"; shows $typLesson$.wWeekdayOff_Minute[15]; editable 0..59
rectangle at (689,34)-(734,60): text "15"
rectangle at (689,176)-(734,202): text ":"; tooltip Switch ON time
rectangle at (694,181)-(709,197): text "%0.2d"; shows $typLesson$.wWeekendOn_hour[15]; editable 0..23
rectangle at (714,181)-(729,197): text "%0.2d"; shows $typLesson$.wWeekendOn_Minute[15]; editable 0..59
rectangle at (689,202)-(734,228): text ":"; tooltip Switch OFF time
rectangle at (694,206)-(709,222): text "%0.2d"; shows $typLesson$.wWeekendOff_hour[15]; editable 0..23
rectangle at (714,206)-(729,222): text "%0.2d"; shows $typLesson$.wWeekendOff_Minute[15]; editable 0..59
rectangle at (689,150)-(734,176): text "15"
4 more shapes without text or variables
*)
